C05455=1036.004,-58.740,418.899,168.441,38.908,157.287
C05456=1036.009,-58.491,418.887,168.443,38.908,157.287
C05457=1036.015,-58.241,418.875,168.446,38.907,157.287
C05458=1036.022,-57.992,418.863,168.448,38.907,157.287
C05459=1036.028,-57.742,418.850,168.451,38.906,157.287
C05460=1036.034,-57.492,418.839,168.453,38.906,157.287
C05461=1036.041,-57.242,418.827,168.456,38.906,157.287
C05462=1036.046,-56.993,418.815,168.458,38.905,157.287
C05463=1036.053,-56.743,418.803,168.461,38.905,157.287
C05464=1036.060,-56.494,418.791,168.464,38.904,157.287
C05465=1036.066,-56.248,418.779,168.466,38.904,157.287
C05466=1036.072,-56.003,418.767,168.469,38.904,157.287
C05467=1036.078,-55.758,418.755,168.470,38.903,157.287
C05468=1036.084,-55.512,418.743,168.473,38.903,157.287
C05469=1036.090,-55.268,418.731,168.475,38.902,157.286
C05470=1036.097,-55.022,418.720,168.478,38.902,157.287
C05471=1036.103,-54.777,418.707,168.480,38.902,157.287
C05472=1036.109,-54.531,418.696,168.483,38.901,157.286
C05473=1036.115,-54.282,418.684,168.485,38.901,157.287
C05474=1036.122,-54.032,418.672,168.488,38.901,157.287
C05475=1036.128,-53.782,418.659,168.490,38.900,157.286
C05476=1036.135,-53.533,418.647,168.493,38.900,157.287
C05477=1036.141,-53.283,418.635,168.495,38.899,157.286
C05478=1036.147,-53.033,418.623,168.498,38.899,157.286
C05479=1036.154,-52.784,418.611,168.500,38.899,157.287
C05480=1036.160,-52.534,418.599,168.503,38.898,157.286
C05481=1036.168,-52.244,418.584,168.506,38.898,157.286
C05482=1036.174,-51.954,418.570,168.509,38.897,157.286
C05483=1036.182,-51.664,418.556,168.512,38.897,157.286
C05484=1036.190,-51.373,418.541,168.515,38.896,157.286
C05485=1036.197,-51.124,418.529,168.517,38.896,157.286
C05486=1036.203,-50.874,418.517,168.520,38.895,157.286
C05487=1036.209,-50.624,418.505,168.522,38.895,157.286
C05488=1036.216,-50.375,418.493,168.525,38.894,157.286
C05489=1036.222,-50.125,418.480,168.527,38.894,157.286
C05490=1036.228,-49.876,418.467,168.530,38.894,157.287
C05491=1036.234,-49.626,418.454,168.532,38.894,157.287
C05492=1036.240,-49.377,418.443,168.535,38.894,157.287
C05493=1036.246,-49.127,418.430,168.537,38.893,157.287
C05494=1036.252,-48.878,418.417,168.539,38.893,157.287
C05495=1036.259,-48.628,418.405,168.542,38.893,157.287
C05496=1036.265,-48.378,418.393,168.544,38.893,157.287
C05497=1036.270,-48.129,418.380,168.547,38.892,157.287
C05498=1036.277,-47.880,418.367,168.549,38.892,157.287
C05499=1036.283,-47.630,418.355,168.552,38.892,157.287
C05500=1036.289,-47.380,418.342,168.554,38.892,157.287
C05501=1036.295,-47.131,418.329,168.557,38.891,157.287
C05502=1036.302,-46.881,418.317,168.559,38.891,157.287
C05503=1036.308,-46.631,418.304,168.562,38.891,157.287
C05504=1036.314,-46.382,418.291,168.564,38.891,157.287
C05505=1036.320,-46.132,418.279,168.566,38.891,157.287
C05506=1036.327,-45.882,418.267,168.569,38.890,157.287
C05507=1036.333,-45.633,418.253,168.571,38.890,157.287
C05508=1036.339,-45.383,418.241,168.574,38.889,157.287
C05509=1036.345,-45.134,418.229,168.576,38.889,157.287
C05510=1036.352,-44.884,418.215,168.579,38.889,157.287
C05511=1036.358,-44.634,418.203,168.581,38.889,157.287
C05512=1036.364,-44.385,418.189,168.584,38.889,157.287
C05513=1036.371,-44.135,418.177,168.586,38.889,157.287
C05514=1036.377,-43.885,418.165,168.588,38.889,157.287
C05515=1036.383,-43.636,418.152,168.591,38.888,157.287
C05516=1036.389,-43.386,418.139,168.593,38.888,157.287
C05517=1036.396,-43.137,418.126,168.596,38.887,157.287
C05518=1036.402,-42.887,418.114,168.598,38.887,157.287
C05519=1036.408,-42.638,418.101,168.601,38.887,157.287
C05520=1036.414,-42.388,418.088,168.603,38.887,157.287
C05521=1036.421,-42.139,418.075,168.606,38.887,157.287
C05522=1036.428,-41.888,418.062,168.608,38.887,157.287
C05523=1036.434,-41.639,418.049,168.610,38.887,157.287
C05524=1036.440,-41.389,418.037,168.613,38.886,157.287
C05525=1036.446,-41.140,418.023,168.615,38.886,157.287
C05526=1036.453,-40.890,418.011,168.618,38.885,157.287
C05527=1036.459,-40.641,417.998,168.620,38.885,157.287
C05528=1036.465,-40.391,417.986,168.623,38.885,157.287
C05529=1036.471,-40.141,417.972,168.625,38.885,157.287
C05530=1036.478,-39.892,417.960,168.627,38.885,157.287
C05531=1036.484,-39.642,417.947,168.630,38.885,157.288
C05532=1036.490,-39.393,417.934,168.632,38.885,157.288
C05533=1036.496,-39.143,417.921,168.635,38.884,157.287
C05534=1036.502,-38.893,417.908,168.637,38.884,157.288
C05535=1036.510,-38.644,417.895,168.640,38.883,157.288
C05536=1036.515,-38.394,417.881,168.642,38.883,157.288
C05537=1036.521,-38.144,417.869,168.644,38.883,157.288
C05538=1036.528,-37.895,417.856,168.647,38.883,157.288
C05539=1036.534,-37.646,417.842,168.649,38.883,157.288
C05540=1036.540,-37.396,417.830,168.651,38.883,157.288
C05541=1036.546,-37.146,417.816,168.654,38.883,157.288
C05542=1036.553,-36.897,417.803,168.656,38.883,157.288
C05543=1036.559,-36.647,417.790,168.659,38.883,157.288
C05544=1036.565,-36.398,417.777,168.662,38.883,157.288
C05545=1036.572,-36.117,417.762,168.665,38.883,157.288
C05546=1036.580,-35.835,417.747,168.667,38.882,157.288
C05547=1036.586,-35.554,417.733,168.670,38.882,157.288
C05548=1036.593,-35.273,417.718,168.673,38.882,157.288
C05549=1036.600,-35.024,417.704,168.675,38.882,157.288
C05550=1036.606,-34.774,417.692,168.677,38.882,157.288
C05551=1036.612,-34.524,417.678,168.680,38.882,157.288
C05552=1036.619,-34.275,417.665,168.682,38.882,157.288
C05553=1036.625,-34.026,417.652,168.684,38.881,157.288
C05554=1036.631,-33.776,417.639,168.687,38.881,157.288
C05555=1036.638,-33.526,417.625,168.689,38.881,157.288
C05556=1036.644,-33.277,417.612,168.692,38.881,157.289
C05557=1036.650,-33.027,417.599,168.694,38.881,157.289
C05558=1036.655,-32.778,417.585,168.696,38.881,157.289
C05559=1036.662,-32.528,417.571,168.699,38.880,157.289
C05560=1036.668,-32.278,417.559,168.701,38.880,157.289
C05561=1036.674,-32.029,417.546,168.703,38.880,157.289
C05562=1036.681,-31.780,417.532,168.706,38.880,157.289
C05563=1036.687,-31.530,417.519,168.708,38.880,157.289
C05564=1036.694,-31.280,417.505,168.710,38.880,157.289
C05565=1036.700,-31.031,417.492,168.713,38.880,157.289
C05566=1036.707,-30.781,417.479,168.715,38.880,157.289
C05567=1036.713,-30.532,417.465,168.717,38.880,157.289
C05568=1036.719,-30.283,417.452,168.720,38.880,157.289
C05569=1036.726,-30.032,417.439,168.722,38.880,157.289
C05570=1036.732,-29.783,417.426,168.725,38.880,157.289
C05571=1036.738,-29.533,417.413,168.727,38.879,157.289
C05572=1036.745,-29.283,417.399,168.729,38.879,157.289
C05573=1036.751,-29.034,417.386,168.732,38.879,157.289
C05574=1036.757,-28.785,417.372,168.734,38.879,157.289
C05575=1036.763,-28.535,417.358,168.736,38.879,157.289
C05576=1036.770,-28.285,417.345,168.739,38.879,157.289
C05577=1036.776,-28.036,417.332,168.741,38.879,157.289
C05578=1036.783,-27.786,417.318,168.743,38.878,157.289
C05579=1036.789,-27.537,417.305,168.746,38.878,157.289
C05580=1036.796,-27.287,417.291,168.748,38.878,157.290
C05581=1036.802,-27.038,417.278,168.750,38.878,157.290
C05582=1036.807,-26.788,417.264,168.753,38.878,157.290
C05583=1036.814,-26.538,417.250,168.755,38.878,157.290
C05584=1036.820,-26.289,417.237,168.757,38.878,157.290
C05585=1036.826,-26.039,417.223,168.761,38.878,157.290
C05586=1036.833,-25.789,417.209,168.763,38.878,157.290
C05587=1036.839,-25.541,417.196,168.765,38.878,157.290
C05588=1036.846,-25.291,417.182,168.767,38.878,157.290
C05589=1036.851,-25.041,417.168,168.770,38.878,157.290
C05590=1036.858,-24.792,417.155,168.772,38.878,157.290
C05591=1036.865,-24.542,417.141,168.774,38.878,157.290
C05592=1036.870,-24.292,417.127,168.777,38.878,157.290
C05593=1036.876,-24.043,417.114,168.779,38.878,157.290
C05594=1036.883,-23.793,417.099,168.781,38.878,157.290
C05595=1036.889,-23.544,417.086,168.783,38.878,157.290
C05596=1036.896,-23.294,417.072,168.786,38.878,157.290
C05597=1036.901,-23.045,417.058,168.788,38.878,157.290
C05598=1036.908,-22.795,417.045,168.790,38.878,157.291
C05599=1036.914,-22.546,417.031,168.793,38.878,157.291
C05600=1036.920,-22.296,417.017,168.795,38.878,157.291
C05601=1036.927,-22.046,417.003,168.797,38.878,157.291
C05602=1036.933,-21.797,416.990,168.799,38.878,157.291
C05603=1036.939,-21.548,416.975,168.802,38.877,157.291
C05604=1036.946,-21.298,416.962,168.804,38.878,157.291
C05605=1036.952,-21.048,416.948,168.806,38.878,157.291
C05606=1036.958,-20.799,416.934,168.809,38.878,157.291
C05607=1036.965,-20.549,416.920,168.811,38.878,157.291
C05608=1036.971,-20.300,416.907,168.813,38.877,157.291
C05609=1036.979,-20.018,416.890,168.817,38.878,157.291
C05610=1036.985,-19.736,416.875,168.819,38.878,157.291
C05611=1036.992,-19.454,416.859,168.822,38.878,157.291
C05612=1036.999,-19.172,416.843,168.824,38.877,157.291
C05613=1037.006,-18.923,416.829,168.827,38.877,157.291
C05614=1037.013,-18.673,416.816,168.829,38.878,157.292
C05615=1037.018,-18.424,416.802,168.831,38.878,157.292
C05616=1037.025,-18.174,416.787,168.833,38.878,157.292
C05617=1037.031,-17.925,416.774,168.836,38.877,157.292
C05618=1037.038,-17.675,416.760,168.838,38.877,157.292
C05619=1037.044,-17.426,416.746,168.840,38.877,157.292
C05620=1037.050,-17.176,416.732,168.843,38.878,157.292
C05621=1037.056,-16.927,416.718,168.845,38.877,157.292
C05622=1037.063,-16.677,416.704,168.847,38.877,157.292
C05623=1037.070,-16.427,416.690,168.849,38.877,157.292
C05624=1037.076,-16.178,416.676,168.852,38.877,157.292
C05625=1037.082,-15.928,416.662,168.854,38.878,157.292
C05626=1037.089,-15.680,416.648,168.856,38.877,157.292
C05627=1037.095,-15.430,416.634,168.858,38.877,157.292
C05628=1037.101,-15.180,416.620,168.861,38.877,157.292
C05629=1037.107,-14.930,416.605,168.863,38.878,157.292
C05630=1037.114,-14.681,416.592,168.865,38.877,157.293
C05631=1037.120,-14.431,416.577,168.867,38.877,157.293
C05632=1037.127,-14.182,416.563,168.870,38.878,157.293
C05633=1037.133,-13.933,416.549,168.873,38.878,157.293
C05634=1037.139,-13.683,416.534,168.875,38.878,157.293
C05635=1037.145,-13.434,416.521,168.877,38.878,157.293
C05636=1037.152,-13.184,416.506,168.879,38.878,157.293
C05637=1037.157,-12.934,416.492,168.882,38.878,157.293
C05638=1037.164,-12.685,416.477,168.884,38.878,157.293
C05639=1037.170,-12.435,416.463,168.886,38.878,157.293
C05640=1037.176,-12.186,416.449,168.888,38.878,157.293
C05641=1037.183,-11.936,416.434,168.890,38.879,157.293
C05642=1037.189,-11.687,416.420,168.893,38.878,157.293
C05643=1037.196,-11.438,416.406,168.895,38.878,157.293
C05644=1037.202,-11.188,416.391,168.897,38.878,157.293
C05645=1037.208,-10.938,416.377,168.899,38.879,157.294
C05646=1037.215,-10.689,416.363,168.901,38.879,157.294
C05647=1037.221,-10.439,416.349,168.904,38.878,157.294
C05648=1037.227,-10.190,416.334,168.906,38.879,157.294
C05649=1037.234,-9.940,416.320,168.908,38.879,157.294
C05650=1037.239,-9.691,416.306,168.910,38.879,157.294
C05651=1037.246,-9.441,416.291,168.913,38.879,157.294
C05652=1037.253,-9.192,416.277,168.916,38.879,157.294
C05653=1037.258,-8.943,416.262,168.918,38.879,157.294
C05654=1037.264,-8.693,416.248,168.920,38.879,157.294
C05655=1037.272,-8.443,416.233,168.922,38.879,157.294
C05656=1037.277,-8.194,416.219,168.924,38.879,157.294
C05657=1037.283,-7.944,416.205,168.927,38.880,157.295
C05658=1037.291,-7.695,416.190,168.929,38.880,157.295
C05659=1037.297,-7.445,416.175,168.931,38.879,157.295
C05660=1037.303,-7.196,416.161,168.933,38.880,157.295
C05661=1037.310,-6.946,416.147,168.935,38.880,157.295
C05662=1037.316,-6.696,416.132,168.938,38.880,157.295
C05663=1037.322,-6.447,416.118,168.940,38.880,157.295
C05664=1037.328,-6.198,416.103,168.942,38.880,157.295
C05665=1037.335,-5.948,416.089,168.944,38.880,157.295
C05666=1037.341,-5.698,416.074,168.946,38.880,157.295
C05667=1037.347,-5.449,416.059,168.949,38.880,157.295
C05668=1037.354,-5.200,416.045,168.951,38.880,157.295
C05669=1037.361,-4.950,416.030,168.953,38.880,157.295
C05670=1037.367,-4.701,416.015,168.956,38.881,157.295
C05671=1037.373,-4.451,416.002,168.958,38.880,157.296
C05672=1037.380,-4.202,415.987,168.960,38.880,157.296
C05673=1037.387,-3.918,415.971,168.963,38.881,157.296
C05674=1037.394,-3.635,415.954,168.965,38.881,157.296
C05675=1037.402,-3.351,415.937,168.968,38.881,157.296
C05676=1037.408,-3.067,415.920,168.970,38.881,157.296
C05677=1037.414,-2.818,415.905,168.972,38.881,157.296
C05678=1037.420,-2.569,415.890,168.975,38.881,157.296
C05679=1037.427,-2.319,415.875,168.977,38.882,157.296
C05680=1037.433,-2.069,415.861,168.979,38.882,157.296
C05681=1037.439,-1.820,415.846,168.981,38.882,157.296
C05682=1037.445,-1.571,415.831,168.983,38.882,157.297
C05683=1037.452,-1.321,415.816,168.985,38.883,157.297
C05684=1037.458,-1.071,415.801,168.987,38.882,157.297
C05685=1037.464,-0.823,415.787,168.990,38.883,157.297
C05686=1037.470,-0.573,415.772,168.993,38.883,157.297
C05687=1037.476,-0.323,415.757,168.995,38.883,157.297
C05688=1037.483,-0.074,415.742,168.997,38.883,157.297
C05689=1037.489,0.175,415.727,168.999,38.884,157.297
C05690=1037.495,0.425,415.712,169.001,38.884,157.297
C05691=1037.501,0.675,415.697,169.003,38.884,157.297
C05692=1037.508,0.924,415.682,169.005,38.884,157.297
C05693=1037.514,1.173,415.667,169.007,38.885,157.298
C05694=1037.520,1.422,415.652,169.009,38.884,157.298
C05695=1037.527,1.672,415.637,169.012,38.884,157.298
C05696=1037.533,1.922,415.622,169.014,38.885,157.298
C05697=1037.539,2.171,415.607,169.016,38.885,157.298
C05698=1037.546,2.421,415.592,169.019,38.885,157.298
C05699=1037.552,2.671,415.577,169.021,38.885,157.298
C05700=1037.558,2.920,415.563,169.023,38.886,157.298
C05701=1037.565,3.169,415.547,169.025,38.885,157.298
C05702=1037.571,3.418,415.532,169.027,38.886,157.298
C05703=1037.577,3.668,415.517,169.029,38.886,157.298
C05704=1037.584,3.918,415.502,169.032,38.886,157.299
C05705=1037.590,4.167,415.487,169.034,38.886,157.299
C05706=1037.595,4.417,415.472,169.036,38.887,157.299
C05707=1037.602,4.666,415.456,169.038,38.887,157.299
C05708=1037.608,4.915,415.441,169.040,38.887,157.299
C05709=1037.615,5.165,415.427,169.042,38.887,157.299
C05710=1037.621,5.415,415.412,169.044,38.888,157.299
C05711=1037.627,5.664,415.397,169.046,38.887,157.299
C05712=1037.634,5.913,415.381,169.049,38.888,157.299
C05713=1037.641,6.163,415.366,169.052,38.888,157.299
C05714=1037.647,6.413,415.351,169.054,38.888,157.299
C05715=1037.653,6.662,415.337,169.056,38.888,157.300
C05716=1037.659,6.911,415.321,169.058,38.888,157.300
C05717=1037.666,7.160,415.306,169.060,38.889,157.300
C05718=1037.672,7.410,415.291,169.062,38.888,157.300
C05719=1037.679,7.660,415.276,169.064,38.889,157.300
C05720=1037.685,7.909,415.260,169.066,38.889,157.300
C05721=1037.691,8.159,415.245,169.068,38.889,157.300
C05722=1037.697,8.408,415.230,169.070,38.889,157.300
C05723=1037.704,8.657,415.214,169.073,38.890,157.300
C05724=1037.710,8.907,415.199,169.075,38.890,157.300
C05725=1037.717,9.157,415.184,169.077,38.889,157.300
C05726=1037.723,9.406,415.169,169.080,38.890,157.301
C05727=1037.730,9.655,415.154,169.082,38.890,157.301
C05728=1037.736,9.905,415.139,169.084,38.890,157.301
C05729=1037.743,10.154,415.123,169.086,38.890,157.301
C05730=1037.749,10.404,415.108,169.088,38.891,157.301
C05731=1037.756,10.653,415.093,169.090,38.891,157.301
C05732=1037.762,10.902,415.078,169.092,38.891,157.301
C05733=1037.768,11.152,415.062,169.095,38.891,157.301
C05734=1037.774,11.402,415.047,169.097,38.891,157.301
C05735=1037.781,11.651,415.031,169.099,38.891,157.301
C05736=1037.787,11.901,415.016,169.101,38.891,157.301
C05737=1037.795,12.186,414.999,169.103,38.892,157.301
C05738=1037.802,12.471,414.981,169.106,38.892,157.302
C05739=1037.810,12.757,414.964,169.108,38.892,157.302
C05740=1037.817,13.042,414.946,169.110,38.892,157.302
C05741=1037.824,13.291,414.931,169.114,38.892,157.302
C05742=1037.830,13.541,414.916,169.116,38.892,157.302
C05743=1037.836,13.790,414.900,169.118,38.893,157.302
C05744=1037.843,14.040,414.885,169.120,38.893,157.302
C05745=1037.849,14.289,414.869,169.122,38.893,157.302
C05746=1037.856,14.538,414.854,169.124,38.893,157.302
C05747=1037.862,14.788,414.838,169.126,38.894,157.302
C05748=1037.868,15.037,414.823,169.128,38.893,157.302
C05749=1037.875,15.287,414.807,169.130,38.894,157.303
C05750=1037.880,15.536,414.792,169.132,38.895,157.303
C05751=1037.887,15.786,414.776,169.134,38.894,157.303
C05752=1037.893,16.035,414.760,169.136,38.895,157.303
C05753=1037.899,16.285,414.745,169.138,38.895,157.303
C05754=1037.906,16.534,414.729,169.141,38.895,157.303
C05755=1037.912,16.784,414.714,169.143,38.895,157.303
C05756=1037.918,17.033,414.698,169.145,38.896,157.303
C05757=1037.925,17.282,414.682,169.147,38.896,157.303
C05758=1037.931,17.532,414.667,169.149,38.896,157.304
C05759=1037.937,17.781,414.651,169.151,38.897,157.304
C05760=1037.943,18.030,414.635,169.153,38.896,157.304
C05761=1037.950,18.280,414.619,169.156,38.897,157.304
C05762=1037.957,18.529,414.604,169.158,38.897,157.304
C05763=1037.963,18.779,414.588,169.160,38.897,157.304
C05764=1037.969,19.028,414.573,169.162,38.897,157.304
C05765=1037.976,19.277,414.557,169.164,38.898,157.304
C05766=1037.982,19.527,414.541,169.167,38.898,157.304
C05767=1037.988,19.776,414.526,169.169,38.898,157.304
C05768=1037.994,20.026,414.509,169.171,38.899,157.305
C05769=1038.001,20.275,414.494,169.173,38.899,157.305
C05770=1038.007,20.525,414.478,169.175,38.899,157.305
C05771=1038.014,20.775,414.462,169.177,38.900,157.305
C05772=1038.020,21.024,414.446,169.179,38.899,157.305
C05773=1038.027,21.273,414.430,169.181,38.900,157.305
C05774=1038.033,21.522,414.414,169.183,38.900,157.305
C05775=1038.039,21.772,414.399,169.185,38.900,157.305
C05776=1038.045,22.021,414.383,169.187,38.901,157.305
C05777=1038.052,22.270,414.367,169.189,38.901,157.305
C05778=1038.058,22.520,414.351,169.192,38.901,157.306
C05779=1038.065,22.769,414.335,169.194,38.902,157.306
C05780=1038.071,23.019,414.319,169.196,38.902,157.306
C05781=1038.077,23.268,414.304,169.198,38.902,157.306
C05782=1038.083,23.518,414.287,169.200,38.902,157.306
C05783=1038.090,23.767,414.272,169.202,38.903,157.306
C05784=1038.096,24.016,414.256,169.204,38.903,157.306
C05785=1038.102,24.265,414.239,169.206,38.903,157.306
C05786=1038.109,24.516,414.224,169.208,38.904,157.306
C05787=1038.115,24.765,414.208,169.210,38.903,157.307
C05788=1038.121,25.014,414.192,169.212,38.904,157.307
C05789=1038.127,25.264,414.176,169.215,38.904,157.307
C05790=1038.134,25.513,414.160,169.217,38.904,157.307
C05791=1038.141,25.763,414.144,169.219,38.905,157.307
C05792=1038.147,26.012,414.128,169.221,38.905,157.307
C05793=1038.153,26.261,414.112,169.223,38.905,157.307
C05794=1038.159,26.510,414.095,169.225,38.906,157.307
C05795=1038.166,26.759,414.080,169.227,38.906,157.307
C05796=1038.172,27.009,414.063,169.229,38.906,157.308
C05797=1038.179,27.258,414.047,169.231,38.906,157.308
C05798=1038.185,27.508,414.031,169.233,38.907,157.308
C05799=1038.191,27.758,414.016,169.235,38.907,157.308
C05800=1038.198,28.008,414.000,169.237,38.907,157.308
C05801=1038.205,28.294,413.981,169.240,38.907,157.308
C05802=1038.212,28.580,413.962,169.243,38.908,157.308
C05803=1038.219,28.867,413.944,169.245,38.908,157.308
C05804=1038.226,29.153,413.925,169.247,38.908,157.308
C05805=1038.233,29.404,413.908,169.249,38.909,157.309
C05806=1038.239,29.653,413.892,169.251,38.909,157.309
C05807=1038.246,29.902,413.877,169.253,38.910,157.309
C05808=1038.252,30.151,413.860,169.255,38.910,157.309
C05809=1038.258,30.401,413.844,169.257,38.910,157.309
C05810=1038.264,30.650,413.827,169.260,38.911,157.309
C05811=1038.271,30.899,413.811,169.262,38.911,157.309
C05812=1038.277,31.148,413.795,169.264,38.911,157.309
C05813=1038.284,31.398,413.778,169.266,38.912,157.310
C05814=1038.290,31.648,413.762,169.268,38.912,157.310
C05815=1038.296,31.897,413.746,169.270,38.912,157.310
C05816=1038.302,32.146,413.730,169.272,38.913,157.310
C05817=1038.309,32.396,413.713,169.274,38.912,157.310
C05818=1038.315,32.645,413.696,169.276,38.913,157.310
C05819=1038.321,32.894,413.680,169.278,38.913,157.310
C05820=1038.327,33.144,413.664,169.280,38.913,157.310
C05821=1038.334,33.393,413.648,169.283,38.914,157.310
C05822=1038.340,33.643,413.632,169.285,38.914,157.311
C05823=1038.346,33.891,413.615,169.287,38.915,157.311
C05824=1038.353,34.142,413.598,169.289,38.915,157.311
C05825=1038.360,34.391,413.582,169.291,38.915,157.311
C05826=1038.366,34.640,413.566,169.293,38.916,157.311
C05827=1038.372,34.890,413.549,169.295,38.916,157.311
C05828=1038.378,35.139,413.533,169.297,38.916,157.311
C05829=1038.384,35.388,413.516,169.299,38.917,157.311
C05830=1038.392,35.638,413.500,169.301,38.917,157.311
C05831=1038.398,35.887,413.484,169.303,38.917,157.312
C05832=1038.404,36.136,413.467,169.305,38.917,157.312
C05833=1038.410,36.386,413.450,169.307,38.918,157.312
C05834=1038.416,36.635,413.434,169.309,38.918,157.312
C05835=1038.422,36.885,413.418,169.311,38.918,157.312
C05836=1038.430,37.134,413.401,169.313,38.918,157.312
C05837=1038.436,37.383,413.385,169.315,38.919,157.312
C05838=1038.442,37.633,413.368,169.317,38.920,157.312
C05839=1038.449,37.882,413.351,169.319,38.919,157.312
C05840=1038.455,38.131,413.335,169.321,38.920,157.313
C05841=1038.461,38.381,413.318,169.323,38.920,157.313
C05842=1038.467,38.630,413.301,169.326,38.921,157.313
C05843=1038.473,38.879,413.285,169.328,38.921,157.313
C05844=1038.480,39.129,413.268,169.330,38.921,157.313
C05845=1038.486,39.378,413.252,169.332,38.922,157.313
C05846=1038.492,39.627,413.235,169.334,38.922,157.313
C05847=1038.499,39.877,413.218,169.336,38.922,157.313
C05848=1038.505,40.126,413.202,169.338,38.923,157.314
C05849=1038.512,40.376,413.184,169.340,38.923,157.314
C05850=1038.517,40.625,413.168,169.342,38.924,157.314
C05851=1038.523,40.874,413.151,169.344,38.924,157.314
C05852=1038.530,41.124,413.134,169.346,38.924,157.314
C05853=1038.536,41.373,413.118,169.348,38.925,157.314
C05854=1038.543,41.623,413.100,169.350,38.925,157.314
C05855=1038.549,41.872,413.084,169.352,38.926,157.315
C05856=1038.555,42.121,413.067,169.354,38.926,157.315
C05857=1038.561,42.371,413.050,169.356,38.926,157.315
C05858=1038.568,42.620,413.034,169.358,38.927,157.315
C05859=1038.574,42.870,413.017,169.360,38.927,157.315
C05860=1038.581,43.119,413.000,169.362,38.927,157.315
C05861=1038.586,43.368,412.984,169.365,38.928,157.315
C05862=1038.593,43.617,412.966,169.367,38.928,157.315
C05863=1038.599,43.866,412.949,169.369,38.929,157.315
C05864=1038.605,44.116,412.932,169.370,38.929,157.316
C05865=1038.612,44.403,412.913,169.373,38.930,157.316
C05866=1038.619,44.689,412.893,169.375,38.930,157.316
C05867=1038.626,44.976,412.873,169.377,38.931,157.316
C05868=1038.634,45.262,412.854,169.379,38.931,157.316
C05869=1038.640,45.512,412.837,169.382,38.932,157.316
C05870=1038.646,45.761,412.820,169.384,38.932,157.317
C05871=1038.653,46.010,412.802,169.386,38.932,157.317
C05872=1038.658,46.260,412.786,169.388,38.933,157.317
C05873=1038.664,46.509,412.769,169.390,38.933,157.317
C05874=1038.671,46.758,412.751,169.392,38.934,157.317
C05875=1038.676,47.008,412.734,169.394,38.934,157.317
C05876=1038.683,47.257,412.717,169.395,38.935,157.317
C05877=1038.690,47.506,412.700,169.398,38.935,157.318
C05878=1038.695,47.756,412.683,169.400,38.935,157.318
C05879=1038.702,48.005,412.666,169.402,38.936,157.318
C05880=1038.708,48.254,412.649,169.404,38.936,157.318
C05881=1038.715,48.503,412.632,169.406,38.937,157.318
C05882=1038.721,48.754,412.614,169.408,38.937,157.318
C05883=1038.727,49.002,412.597,169.410,38.938,157.318
C05884=1038.734,49.252,412.580,169.412,38.938,157.318
C05885=1038.739,49.501,412.563,169.414,38.938,157.319
C05886=1038.746,49.751,412.546,169.416,38.939,157.319
C05887=1038.752,50.000,412.529,169.418,38.939,157.319
C05888=1038.758,50.249,412.511,169.420,38.940,157.319
C05889=1038.764,50.498,412.494,169.422,38.940,157.319
C05890=1038.771,50.748,412.477,169.424,38.941,157.319
C05891=1038.776,50.997,412.460,169.426,38.941,157.319
C05892=1038.783,51.247,412.443,169.428,38.941,157.319
C05893=1038.790,51.495,412.426,169.430,38.942,157.320
C05894=1038.796,51.745,412.408,169.432,38.942,157.320
C05895=1038.802,51.994,412.391,169.435,38.943,157.320
C05896=1038.808,52.244,412.374,169.436,38.943,157.320
C05897=1038.814,52.493,412.356,169.438,38.943,157.320
C05898=1038.821,52.742,412.339,169.440,38.944,157.320
C05899=1038.828,52.992,412.322,169.442,38.944,157.320
C05900=1038.833,53.241,412.304,169.444,38.945,157.321
C05901=1038.840,53.490,412.287,169.446,38.945,157.321
C05902=1038.845,53.740,412.270,169.448,38.945,157.321
C05903=1038.852,53.989,412.253,169.450,38.946,157.321
C05904=1038.858,54.238,412.236,169.453,38.946,157.321
C05905=1038.865,54.488,412.218,169.455,38.947,157.321
C05906=1038.871,54.737,412.200,169.457,38.947,157.321
C05907=1038.878,54.986,412.183,169.458,38.947,157.321
C05908=1038.884,55.236,412.166,169.460,38.948,157.322
C05909=1038.890,55.484,412.149,169.462,38.948,157.322
C05910=1038.897,55.734,412.131,169.464,38.949,157.322
C05911=1038.903,55.984,412.113,169.466,38.949,157.322
C05912=1038.909,56.232,412.096,169.468,38.949,157.322
C05913=1038.916,56.482,412.079,169.471,38.949,157.322
C05914=1038.922,56.731,412.061,169.473,38.950,157.322
C05915=1038.929,56.980,412.044,169.475,38.950,157.322
C05916=1038.934,57.231,412.027,169.477,38.951,157.323
C05917=1038.941,57.479,412.010,169.479,38.951,157.323
C05918=1038.947,57.729,411.993,169.480,38.951,157.323
C05919=1038.954,57.978,411.975,169.482,38.952,157.323
C05920=1038.960,58.227,411.958,169.484,38.952,157.323
C05921=1038.967,58.477,411.940,169.486,38.952,157.323
C05922=1038.973,58.726,411.922,169.488,38.953,157.323
C05923=1038.979,58.974,411.905,169.491,38.953,157.323
C05924=1038.985,59.224,411.887,169.493,38.954,157.324
C05925=1038.992,59.474,411.869,169.495,38.954,157.324
C05926=1038.999,59.723,411.852,169.497,38.954,157.324
C05927=1039.005,59.972,411.834,169.499,38.955,157.324
C05928=1039.012,60.221,411.817,169.501,38.955,157.324
C05929=1039.019,60.507,411.797,169.503,38.956,157.324
C05930=1039.026,60.794,411.777,169.505,38.956,157.324
C05931=1039.034,61.081,411.757,169.507,38.956,157.324
C05932=1039.041,61.367,411.737,169.510,38.957,157.325
C05933=1039.047,61.616,411.719,169.512,38.957,157.325
C05934=1039.054,61.866,411.701,169.514,38.958,157.325
C05935=1039.060,62.115,411.684,169.516,38.958,157.325
C05936=1039.067,62.364,411.667,169.518,38.958,157.325
C05937=1039.073,62.613,411.648,169.520,38.959,157.325
C05938=1039.080,62.863,411.631,169.522,38.959,157.325
C05939=1039.086,63.112,411.613,169.524,38.959,157.325
C05940=1039.092,63.361,411.596,169.526,38.959,157.326
C05941=1039.099,63.610,411.579,169.529,38.960,157.326
C05942=1039.105,63.860,411.561,169.531,38.961,157.326
C05943=1039.111,64.109,411.543,169.533,38.961,157.326
C05944=1039.118,64.358,411.525,169.534,38.961,157.326
C05945=1039.124,64.608,411.507,169.536,38.961,157.326
C05946=1039.130,64.857,411.489,169.538,38.962,157.326
C05947=1039.137,65.106,411.472,169.540,38.963,157.327
C05948=1039.143,65.355,411.454,169.542,38.963,157.327
C05949=1039.149,65.605,411.436,169.544,38.964,157.327
C05950=1039.155,65.854,411.419,169.547,38.964,157.327
C05951=1039.162,66.103,411.400,169.549,38.965,157.327
C05952=1039.168,66.353,411.382,169.551,38.965,157.327
C05953=1039.175,66.602,411.365,169.552,38.965,157.327
C05954=1039.181,66.851,411.346,169.554,38.965,157.328
C05955=1039.187,67.100,411.329,169.556,38.966,157.328
C05956=1039.194,67.350,411.311,169.558,38.967,157.328
C05957=1039.200,67.599,411.293,169.560,38.967,157.328
C05958=1039.206,67.849,411.275,169.563,38.968,157.328
C05959=1039.212,68.098,411.257,169.565,38.968,157.328
C05960=1039.219,68.346,411.239,169.567,38.969,157.328
C05961=1039.225,68.596,411.221,169.568,38.968,157.328
C05962=1039.231,68.845,411.203,169.570,38.969,157.329
C05963=1039.237,69.095,411.185,169.572,38.970,157.329
C05964=1039.244,69.344,411.168,169.574,38.970,157.329
C05965=1039.250,69.593,411.149,169.576,38.971,157.329
C05966=1039.256,69.843,411.131,169.579,38.971,157.329
C05967=1039.263,70.092,411.112,169.581,38.972,157.329
C05968=1039.268,70.341,411.095,169.583,38.972,157.330
C05969=1039.275,70.590,411.076,169.584,38.973,157.330
C05970=1039.281,70.839,411.059,169.586,38.973,157.330
C05971=1039.288,71.088,411.040,169.588,38.974,157.330
C05972=1039.294,71.338,411.022,169.590,38.974,157.330
C05973=1039.300,71.587,411.005,169.592,38.975,157.330
C05974=1039.306,71.836,410.986,169.595,38.975,157.330
C05975=1039.312,72.085,410.967,169.597,38.975,157.330
C05976=1039.319,72.335,410.950,169.599,38.976,157.331
C05977=1039.325,72.584,410.931,169.600,38.976,157.331
C05978=1039.332,72.834,410.914,169.602,38.977,157.331
C05979=1039.338,73.082,410.895,169.604,38.977,157.331
C05980=1039.344,73.332,410.877,169.606,38.978,157.331
C05981=1039.350,73.581,410.859,169.608,38.978,157.331
C05982=1039.356,73.831,410.841,169.611,38.979,157.332
C05983=1039.363,74.080,410.822,169.613,38.979,157.332
C05984=1039.369,74.330,410.804,169.615,38.980,157.332
C05985=1039.375,74.578,410.786,169.616,38.980,157.332
C05986=1039.381,74.827,410.767,169.618,38.981,157.332
C05987=1039.387,75.077,410.749,169.620,38.981,157.332
C05988=1039.394,75.326,410.731,169.622,38.982,157.332
C05989=1039.400,75.576,410.713,169.624,38.982,157.333
C05990=1039.407,75.825,410.695,169.626,38.982,157.333
C05991=1039.413,76.074,410.676,169.629,38.983,157.333
C05992=1039.419,76.323,410.658,169.631,38.983,157.333
C05993=1039.426,76.609,410.637,169.633,38.984,157.333
C05994=1039.434,76.895,410.616,169.635,38.984,157.333
C05995=1039.441,77.181,410.594,169.637,38.985,157.333
C05996=1039.448,77.467,410.573,169.639,38.985,157.334
C05997=1039.454,77.716,410.556,169.641,38.986,157.334
C05998=1039.461,77.966,410.537,169.644,38.986,157.334
C05999=1039.467,78.215,410.518,169.646,38.987,157.334
C06000=1039.473,78.465,410.500,169.648,38.987,157.334
C06001=1039.479,78.714,410.481,169.650,38.988,157.334
C06002=1039.485,78.963,410.462,169.651,38.988,157.335
C06003=1039.492,79.212,410.444,169.653,38.989,157.335
C06004=1039.498,79.461,410.426,169.655,38.990,157.335
C06005=1039.504,79.710,410.408,169.658,38.990,157.335
C06006=1039.510,79.960,410.388,169.660,38.991,157.335
C06007=1039.516,80.209,410.370,169.662,38.992,157.335
C06008=1039.522,80.458,410.351,169.664,38.992,157.336
C06009=1039.529,80.707,410.332,169.665,38.993,157.336
C06010=1039.535,80.957,410.314,169.667,38.993,157.336
C06011=1039.541,81.206,410.296,169.669,38.994,157.336
C06012=1039.547,81.455,410.277,169.672,38.994,157.336
C06013=1039.553,81.705,410.258,169.674,38.995,157.336
C06014=1039.560,81.954,410.239,169.676,38.995,157.337
C06015=1039.566,82.203,410.221,169.678,38.996,157.337
C06016=1039.573,82.452,410.202,169.679,38.996,157.337
C06017=1039.578,82.701,410.184,169.681,38.997,157.337
C06018=1039.584,82.950,410.165,169.683,38.997,157.337
C06019=1039.590,83.199,410.146,169.686,38.998,157.337
C06020=1039.597,83.449,410.128,169.688,38.998,157.337
C06021=1039.603,83.698,410.109,169.690,38.999,157.338
C06022=1039.609,83.947,410.090,169.692,38.999,157.338
C06023=1039.615,84.196,410.071,169.694,39.000,157.338
C06024=1039.622,84.445,410.053,169.695,39.000,157.338
C06025=1039.628,84.695,410.034,169.697,39.001,157.338
C06026=1039.635,84.944,410.015,169.699,39.001,157.338
C06027=1039.640,85.193,409.996,169.702,39.002,157.339
C06028=1039.647,85.442,409.977,169.704,39.002,157.339
C06029=1039.653,85.691,409.959,169.706,39.003,157.339
C06030=1039.660,85.940,409.940,169.708,39.003,157.339
C06031=1039.666,86.190,409.922,169.710,39.004,157.339
C06032=1039.671,86.440,409.903,169.711,39.004,157.339
C06033=1039.678,86.689,409.884,169.713,39.005,157.339
C06034=1039.685,86.937,409.865,169.716,39.005,157.340
C06035=1039.692,87.187,409.846,169.718,39.005,157.340
C06036=1039.697,87.436,409.827,169.720,39.006,157.340
C06037=1039.704,87.686,409.808,169.722,39.006,157.340
C06038=1039.710,87.935,409.789,169.724,39.007,157.340
C06039=1039.717,88.184,409.771,169.726,39.007,157.340
C06040=1039.723,88.433,409.752,169.728,39.008,157.340
C06041=1039.729,88.682,409.733,169.729,39.008,157.341
C06042=1039.735,88.932,409.714,169.731,39.009,157.341
C06043=1039.742,89.181,409.696,169.734,39.009,157.341
C06044=1039.748,89.430,409.677,169.736,39.010,157.341
C06045=1039.754,89.679,409.658,169.738,39.010,157.341
C06046=1039.760,89.928,409.639,169.740,39.011,157.341
C06047=1039.766,90.177,409.620,169.742,39.011,157.341
C06048=1039.772,90.427,409.601,169.744,39.012,157.342
C06049=1039.779,90.675,409.582,169.746,39.012,157.342
C06050=1039.785,90.926,409.562,169.748,39.013,157.342
C06051=1039.792,91.175,409.544,169.750,39.014,157.342
C06052=1039.797,91.424,409.524,169.752,39.015,157.342
C06053=1039.804,91.673,409.506,169.754,39.015,157.343
C06054=1039.810,91.922,409.486,169.756,39.016,157.343
C06055=1039.816,92.171,409.467,169.758,39.016,157.343
C06056=1039.822,92.421,409.448,169.760,39.017,157.343
C06057=1039.829,92.707,409.426,169.763,39.017,157.343
C06058=1039.836,92.993,409.404,169.765,39.018,157.343
C06059=1039.844,93.279,409.382,169.767,39.019,157.344
C06060=1039.850,93.564,409.360,169.769,39.019,157.344
C06061=1039.857,93.814,409.341,169.771,39.020,157.344
C06062=1039.863,94.063,409.322,169.773,39.020,157.344
C06063=1039.869,94.312,409.302,169.776,39.021,157.344
C06064=1039.876,94.561,409.283,169.778,39.021,157.344
C06065=1039.881,94.811,409.264,169.780,39.022,157.345
C06066=1039.888,95.059,409.245,169.781,39.022,157.345
C06067=1039.894,95.308,409.225,169.783,39.023,157.345
C06068=1039.900,95.558,409.207,169.785,39.023,157.345
C06069=1039.907,95.807,409.187,169.787,39.024,157.345
C06070=1039.913,96.056,409.168,169.790,39.025,157.345
C06071=1039.919,96.306,409.149,169.792,39.026,157.346
C06072=1039.925,96.554,409.129,169.794,39.026,157.346
C06073=1039.931,96.804,409.110,169.796,39.027,157.346
C06074=1039.937,97.053,409.091,169.797,39.027,157.346
C06075=1039.944,97.302,409.071,169.799,39.028,157.346
C06076=1039.950,97.552,409.052,169.801,39.028,157.346
C06077=1039.956,97.801,409.033,169.804,39.029,157.347
C06078=1039.962,98.050,409.013,169.806,39.029,157.347
C06079=1039.969,98.299,408.995,169.808,39.030,157.347
C06080=1039.975,98.548,408.975,169.810,39.030,157.347
C06081=1039.982,98.797,408.956,169.812,39.031,157.347
C06082=1039.987,99.047,408.936,169.814,39.031,157.347
C06083=1039.994,99.295,408.917,169.816,39.032,157.347
C06084=1040.000,99.545,408.898,169.818,39.032,157.348
C06085=1040.007,99.793,408.878,169.820,39.033,157.348
C06086=1040.013,100.043,408.859,169.822,39.033,157.348
C06087=1040.019,100.292,408.839,169.824,39.034,157.348
C06088=1040.025,100.541,408.820,169.826,39.034,157.348
C06089=1040.031,100.790,408.800,169.828,39.035,157.349
C06090=1040.037,101.040,408.781,169.830,39.036,157.349
C06091=1040.044,101.289,408.761,169.833,39.036,157.349
C06092=1040.050,101.538,408.742,169.834,39.037,157.349
C06093=1040.056,101.787,408.722,169.836,39.037,157.349
C06094=1040.062,102.036,408.702,169.838,39.038,157.349
C06095=1040.068,102.285,408.683,169.840,39.039,157.350
C06096=1040.074,102.535,408.662,169.842,39.040,157.350
C06097=1040.081,102.784,408.644,169.845,39.040,157.350
C06098=1040.087,103.033,408.624,169.847,39.041,157.350
C06099=1040.092,103.282,408.605,169.849,39.041,157.350
C06100=1040.099,103.532,408.584,169.851,39.042,157.350
C06101=1040.105,103.780,408.564,169.852,39.043,157.351
C06102=1040.111,104.030,408.545,169.854,39.043,157.351
C06103=1040.117,104.278,408.526,169.856,39.044,157.351
C06104=1040.123,104.527,408.506,169.859,39.044,157.351
C06105=1040.130,104.777,408.486,169.861,39.045,157.351
C06106=1040.136,105.026,408.466,169.863,39.045,157.351
C06107=1040.142,105.275,408.446,169.865,39.046,157.352
C06108=1040.149,105.525,408.427,169.867,39.047,157.352
C06109=1040.155,105.774,408.407,169.869,39.047,157.352
C06110=1040.161,106.022,408.387,169.871,39.048,157.352
C06111=1040.166,106.272,408.368,169.873,39.048,157.352
C06112=1040.173,106.521,408.348,169.875,39.049,157.352
C06113=1040.179,106.770,408.328,169.877,39.049,157.353
C06114=1040.186,107.019,408.308,169.879,39.050,157.353
C06115=1040.192,107.269,408.289,169.881,39.050,157.353
C06116=1040.198,107.518,408.269,169.883,39.052,157.353
C06117=1040.204,107.766,408.249,169.886,39.052,157.353
C06118=1040.210,108.015,408.229,169.888,39.053,157.354
C06119=1040.216,108.265,408.209,169.890,39.053,157.354
C06120=1040.223,108.514,408.190,169.892,39.054,157.354
C06121=1040.230,108.800,408.167,169.894,39.054,157.354
C06122=1040.237,109.086,408.145,169.896,39.055,157.354
C06123=1040.244,109.372,408.121,169.899,39.056,157.354
C06124=1040.251,109.658,408.098,169.901,39.056,157.355
C06125=1040.258,109.907,408.079,169.903,39.057,157.355
C06126=1040.264,110.156,408.059,169.905,39.057,157.355
C06127=1040.270,110.405,408.039,169.907,39.058,157.355
C06128=1040.276,110.654,408.019,169.909,39.059,157.355
C06129=1040.283,110.904,407.999,169.912,39.059,157.356
C06130=1040.289,111.153,407.979,169.914,39.060,157.356
C06131=1040.295,111.402,407.959,169.916,39.060,157.356
C06132=1040.301,111.651,407.939,169.918,39.061,157.356
C06133=1040.307,111.900,407.919,169.920,39.062,157.356
C06134=1040.313,112.149,407.899,169.921,39.063,157.356
C06135=1040.320,112.398,407.879,169.923,39.063,157.357
C06136=1040.326,112.647,407.859,169.926,39.064,157.357
C06137=1040.332,112.896,407.839,169.928,39.064,157.357
C06138=1040.338,113.146,407.818,169.930,39.065,157.357
C06139=1040.344,113.394,407.799,169.932,39.066,157.357
C06140=1040.351,113.644,407.778,169.934,39.066,157.357
C06141=1040.357,113.893,407.758,169.936,39.067,157.358
C06142=1040.362,114.142,407.738,169.939,39.068,157.358
C06143=1040.369,114.391,407.717,169.941,39.068,157.358
C06144=1040.375,114.640,407.697,169.943,39.069,157.358
C06145=1040.381,114.889,407.677,169.944,39.070,157.359
C06146=1040.387,115.139,407.657,169.946,39.071,157.359
C06147=1040.393,115.388,407.637,169.948,39.071,157.359
C06148=1040.399,115.636,407.617,169.951,39.071,157.359
C06149=1040.405,115.886,407.596,169.953,39.073,157.359
C06150=1040.411,116.135,407.576,169.955,39.073,157.359
C06151=1040.417,116.384,407.556,169.957,39.074,157.360
C06152=1040.423,116.633,407.535,169.959,39.075,157.360
C06153=1040.429,116.882,407.514,169.962,39.075,157.360
C06154=1040.435,117.131,407.494,169.964,39.076,157.360
C06155=1040.441,117.380,407.474,169.965,39.077,157.360
C06156=1040.447,117.629,407.454,169.967,39.077,157.361
C06157=1040.453,117.879,407.433,169.969,39.078,157.361
C06158=1040.459,118.128,407.413,169.971,39.078,157.361
C06159=1040.466,118.377,407.393,169.974,39.080,157.361
C06160=1040.471,118.626,407.371,169.976,39.080,157.361
C06161=1040.478,118.875,407.351,169.978,39.081,157.362
C06162=1040.484,119.124,407.331,169.980,39.082,157.362
C06163=1040.490,119.373,407.311,169.982,39.082,157.362
C06164=1040.496,119.623,407.290,169.984,39.083,157.362
C06165=1040.502,119.871,407.270,169.987,39.084,157.362
C06166=1040.509,120.120,407.249,169.989,39.084,157.363
C06167=1040.514,120.369,407.229,169.990,39.085,157.363
C06168=1040.521,120.619,407.208,169.992,39.085,157.363
C06169=1040.527,120.867,407.188,169.994,39.086,157.363
C06170=1040.533,121.117,407.167,169.996,39.087,157.363
C06171=1040.539,121.366,407.147,169.999,39.087,157.363
C06172=1040.545,121.615,407.127,170.001,39.088,157.364
C06173=1040.552,121.864,407.106,170.003,39.089,157.364
C06174=1040.557,122.113,407.085,170.005,39.090,157.364
C06175=1040.563,122.362,407.065,170.007,39.090,157.364
C06176=1040.570,122.612,407.045,170.010,39.091,157.365
C06177=1040.576,122.860,407.023,170.012,39.092,157.365
C06178=1040.582,123.110,407.003,170.014,39.092,157.365
C06179=1040.588,123.359,406.983,170.016,39.093,157.365
C06180=1040.594,123.608,406.961,170.018,39.094,157.365
C06181=1040.600,123.857,406.942,170.020,39.094,157.365
C06182=1040.607,124.106,406.921,170.022,39.095,157.366
C06183=1040.612,124.355,406.900,170.025,39.095,157.366
C06184=1040.619,124.604,406.880,170.027,39.096,157.366
C06185=1040.626,124.889,406.856,170.029,39.097,157.366
C06186=1040.634,125.176,406.832,170.031,39.098,157.366
C06187=1040.640,125.462,406.809,170.033,39.099,157.367
C06188=1040.647,125.747,406.785,170.037,39.099,157.367
C06189=1040.654,125.996,406.764,170.039,39.100,157.367
C06190=1040.660,126.246,406.743,170.041,39.101,157.367
C06191=1040.666,126.495,406.723,170.043,39.101,157.367
C06192=1040.672,126.744,406.702,170.045,39.102,157.368
C06193=1040.678,126.993,406.682,170.048,39.103,157.368
C06194=1040.685,127.241,406.661,170.049,39.103,157.368
C06195=1040.690,127.491,406.640,170.051,39.104,157.368
C06196=1040.697,127.739,406.619,170.053,39.104,157.368
C06197=1040.704,127.989,406.599,170.055,39.105,157.369
C06198=1040.710,128.237,406.578,170.057,39.106,157.369
C06199=1040.716,128.487,406.557,170.059,39.106,157.369
C06200=1040.723,128.736,406.536,170.062,39.107,157.369
C06201=1040.728,128.985,406.516,170.064,39.108,157.369
C06202=1040.735,129.234,406.495,170.066,39.108,157.370
C06203=1040.741,129.483,406.475,170.068,39.109,157.370
C06204=1040.747,129.732,406.453,170.070,39.109,157.370
C06205=1040.754,129.981,406.433,170.073,39.111,157.370
C06206=1040.760,130.230,406.412,170.075,39.111,157.370
C06207=1040.766,130.479,406.391,170.077,39.112,157.370
C06208=1040.773,130.728,406.370,170.079,39.112,157.371
C06209=1040.779,130.977,406.350,170.081,39.113,157.371
C06210=1040.785,131.226,406.328,170.083,39.114,157.371
C06211=1040.791,131.476,406.307,170.085,39.114,157.371
C06212=1040.797,131.724,406.287,170.088,39.115,157.372
C06213=1040.803,131.974,406.265,170.090,39.116,157.372
C06214=1040.809,132.223,406.244,170.092,39.117,157.372
C06215=1040.816,132.472,406.224,170.094,39.117,157.372
C06216=1040.822,132.721,406.202,170.096,39.118,157.372
C06217=1040.828,132.970,406.180,170.099,39.119,157.373
C06218=1040.834,133.219,406.160,170.101,39.120,157.373
C06219=1040.840,133.468,406.139,170.103,39.121,157.373
C06220=1040.846,133.717,406.117,170.105,39.121,157.373
C06221=1040.852,133.966,406.097,170.107,39.122,157.373
C06222=1040.858,134.215,406.076,170.110,39.123,157.374
C06223=1040.864,134.464,406.054,170.112,39.123,157.374
C06224=1040.871,134.713,406.033,170.114,39.124,157.374
C06225=1040.877,134.962,406.012,170.116,39.125,157.374
C06226=1040.883,135.212,405.991,170.118,39.125,157.374
C06227=1040.889,135.460,405.970,170.121,39.126,157.375
C06228=1040.895,135.709,405.948,170.123,39.127,157.375
C06229=1040.902,135.958,405.927,170.125,39.127,157.375
C06230=1040.908,136.207,405.907,170.127,39.129,157.375
C06231=1040.914,136.456,405.885,170.129,39.129,157.375
C06232=1040.920,136.706,405.864,170.132,39.130,157.376
C06233=1040.926,136.954,405.843,170.134,39.131,157.376
C06234=1040.932,137.203,405.821,170.136,39.131,157.376
C06235=1040.938,137.452,405.800,170.138,39.132,157.376
C06236=1040.944,137.702,405.779,170.140,39.133,157.376
C06237=1040.951,137.950,405.758,170.142,39.134,157.377
C06238=1040.957,138.199,405.736,170.145,39.134,157.377
C06239=1040.963,138.449,405.715,170.147,39.136,157.377
C06240=1040.969,138.698,405.693,170.149,39.136,157.377
C06241=1040.975,138.946,405.672,170.151,39.136,157.378
C06242=1040.982,139.195,405.651,170.154,39.138,157.378
C06243=1040.988,139.444,405.629,170.157,39.138,157.378
C06244=1040.994,139.694,405.607,170.159,39.139,157.378
C06245=1040.999,139.942,405.586,170.161,39.140,157.378
C06246=1041.006,140.191,405.565,170.163,39.141,157.379
C06247=1041.012,140.440,405.543,170.165,39.141,157.379
C06248=1041.018,140.690,405.521,170.168,39.142,157.379
C06249=1041.025,140.975,405.498,170.170,39.143,157.379
C06250=1041.032,141.261,405.472,170.172,39.144,157.380
C06251=1041.038,141.547,405.448,170.175,39.145,157.380
C06252=1041.046,141.832,405.423,170.178,39.146,157.380
C06253=1041.052,142.081,405.402,170.180,39.147,157.380
C06254=1041.058,142.330,405.380,170.182,39.148,157.381
C06255=1041.064,142.579,405.359,170.184,39.148,157.381
C06256=1041.070,142.828,405.337,170.186,39.149,157.381
C06257=1041.077,143.077,405.316,170.189,39.150,157.381
C06258=1041.082,143.326,405.294,170.191,39.151,157.382
C06259=1041.089,143.574,405.272,170.193,39.151,157.382
C06260=1041.095,143.824,405.250,170.195,39.153,157.382
C06261=1041.101,144.073,405.229,170.197,39.153,157.382
C06262=1041.107,144.322,405.207,170.200,39.154,157.382
C06263=1041.113,144.571,405.186,170.202,39.155,157.383
C06264=1041.119,144.820,405.164,170.204,39.156,157.383
C06265=1041.125,145.069,405.142,170.206,39.156,157.383
C06266=1041.131,145.318,405.121,170.209,39.157,157.383
C06267=1041.138,145.567,405.098,170.212,39.158,157.384
C06268=1041.144,145.816,405.077,170.214,39.158,157.384
C06269=1041.151,146.065,405.056,170.216,39.159,157.384
C06270=1041.156,146.313,405.035,170.218,39.160,157.384
C06271=1041.162,146.563,405.013,170.220,39.161,157.384
C06272=1041.169,146.811,404.991,170.223,39.161,157.385
C06273=1041.175,147.060,404.969,170.225,39.163,157.385
C06274=1041.181,147.310,404.947,170.227,39.164,157.385
C06275=1041.187,147.559,404.925,170.229,39.164,157.385
C06276=1041.193,147.808,404.903,170.231,39.165,157.386
C06277=1041.199,148.057,404.881,170.234,39.166,157.386
C06278=1041.205,148.305,404.860,170.236,39.167,157.386
C06279=1041.211,148.555,404.838,170.238,39.167,157.386
C06280=1041.217,148.803,404.816,170.240,39.169,157.386
C06281=1041.224,149.052,404.794,170.244,39.170,157.387
C06282=1041.230,149.302,404.773,170.246,39.170,157.387
C06283=1041.235,149.551,404.750,170.248,39.171,157.387
C06284=1041.242,149.800,404.728,170.250,39.172,157.387
C06285=1041.248,150.049,404.706,170.252,39.173,157.388
C06286=1041.254,150.298,404.684,170.255,39.174,157.388
C06287=1041.260,150.546,404.663,170.257,39.174,157.388
C06288=1041.266,150.795,404.640,170.259,39.175,157.388
C06289=1041.272,151.044,404.618,170.261,39.176,157.389
C06290=1041.278,151.293,404.596,170.263,39.177,157.389
C06291=1041.284,151.542,404.574,170.266,39.178,157.389
C06292=1041.291,151.791,404.552,170.268,39.179,157.389
C06293=1041.296,152.040,404.530,170.271,39.180,157.390
C06294=1041.302,152.289,404.508,170.273,39.180,157.390
C06295=1041.309,152.538,404.486,170.276,39.181,157.390
C06296=1041.315,152.787,404.464,170.278,39.182,157.390
C06297=1041.322,153.036,404.442,170.280,39.183,157.391
C06298=1041.327,153.285,404.419,170.282,39.184,157.391
C06299=1041.333,153.534,404.397,170.284,39.185,157.391
C06300=1041.340,153.783,404.375,170.287,39.186,157.391
C06301=1041.346,154.031,404.353,170.289,39.187,157.392
C06302=1041.351,154.281,404.331,170.291,39.187,157.392
C06303=1041.358,154.530,404.308,170.294,39.188,157.392
C06304=1041.364,154.779,404.287,170.297,39.189,157.392
C06305=1041.371,155.027,404.264,170.299,39.190,157.392
C06306=1041.375,155.276,404.243,170.301,39.191,157.393
C06307=1041.382,155.525,404.220,170.303,39.192,157.393
C06308=1041.388,155.774,404.197,170.305,39.193,157.393
C06309=1041.394,156.023,404.176,170.308,39.194,157.393
C06310=1041.400,156.271,404.153,170.310,39.195,157.394
C06311=1041.406,156.520,404.130,170.312,39.196,157.394
C06312=1041.412,156.770,404.109,170.315,39.196,157.394
C06313=1041.420,157.055,404.083,170.318,39.197,157.395
C06314=1041.427,157.341,404.057,170.320,39.199,157.395
C06315=1041.433,157.626,404.032,170.323,39.200,157.395
C06316=1041.440,157.911,404.006,170.325,39.201,157.395
C06317=1041.447,158.160,403.983,170.329,39.202,157.396
C06318=1041.453,158.409,403.962,170.331,39.202,157.396
C06319=1041.458,158.658,403.939,170.333,39.203,157.396
C06320=1041.465,158.906,403.916,170.335,39.204,157.396
C06321=1041.471,159.156,403.895,170.337,39.205,157.397
C06322=1041.477,159.404,403.872,170.340,39.206,157.397
C06323=1041.483,159.653,403.850,170.342,39.207,157.397
C06324=1041.489,159.902,403.827,170.345,39.208,157.397
C06325=1041.496,160.152,403.805,170.347,39.209,157.398
C06326=1041.502,160.401,403.782,170.350,39.210,157.398
C06327=1041.508,160.649,403.759,170.352,39.211,157.398
C06328=1041.514,160.898,403.736,170.354,39.212,157.399
C06329=1041.519,161.147,403.713,170.356,39.213,157.399
C06330=1041.525,161.396,403.690,170.359,39.214,157.399
C06331=1041.531,161.645,403.667,170.361,39.215,157.399
C06332=1041.537,161.893,403.645,170.364,39.216,157.400
C06333=1041.543,162.142,403.622,170.366,39.217,157.400
C06334=1041.549,162.392,403.600,170.369,39.218,157.400
C06335=1041.554,162.641,403.577,170.371,39.219,157.400
C06336=1041.561,162.889,403.555,170.373,39.220,157.401
C06337=1041.566,163.138,403.532,170.376,39.221,157.401
C06338=1041.572,163.387,403.509,170.378,39.222,157.401
C06339=1041.578,163.636,403.486,170.380,39.223,157.402
C06340=1041.584,163.885,403.463,170.383,39.225,157.402
C06341=1041.590,164.134,403.441,170.386,39.226,157.402
C06342=1041.596,164.382,403.418,170.388,39.227,157.403
C06343=1041.602,164.631,403.395,170.390,39.228,157.403
C06344=1041.607,164.880,403.372,170.392,39.228,157.403
C06345=1041.613,165.129,403.349,170.395,39.229,157.403
C06346=1041.620,165.378,403.326,170.398,39.230,157.404
C06347=1041.626,165.627,403.302,170.400,39.232,157.404
C06348=1041.632,165.876,403.279,170.402,39.233,157.404
C06349=1041.638,166.125,403.256,170.405,39.234,157.404
C06350=1041.643,166.373,403.234,170.407,39.235,157.405
C06351=1041.650,166.622,403.211,170.409,39.236,157.405
C06352=1041.656,166.871,403.188,170.412,39.237,157.405
C06353=1041.661,167.120,403.165,170.415,39.238,157.406
C06354=1041.668,167.369,403.142,170.417,39.239,157.406
C06355=1041.673,167.618,403.119,170.419,39.240,157.406
C06356=1041.679,167.867,403.096,170.422,39.241,157.406
C06357=1041.686,168.115,403.073,170.424,39.243,157.407
C06358=1041.692,168.364,403.050,170.427,39.243,157.407
C06359=1041.697,168.613,403.027,170.429,39.244,157.407
C06360=1041.704,168.863,403.004,170.431,39.245,157.408
C06361=1041.710,169.104,402.982,170.434,39.246,157.408
C06362=1041.715,169.347,402.959,170.436,39.247,157.408
C06363=1041.721,169.590,402.936,170.438,39.248,157.408
C06364=1041.727,169.832,402.914,170.442,39.250,157.409
C06365=1041.733,170.074,402.891,170.444,39.251,157.409
C06366=1041.739,170.317,402.870,170.446,39.252,157.409
C06367=1041.745,170.560,402.847,170.448,39.253,157.410
C06368=1041.751,170.803,402.824,170.451,39.253,157.410
C06369=1041.757,171.051,402.801,170.453,39.254,157.410
C06370=1041.763,171.299,402.778,170.456,39.255,157.410
C06371=1041.769,171.548,402.755,170.458,39.257,157.411
C06372=1041.775,171.798,402.731,170.461,39.258,157.411
C06373=1041.781,172.047,402.708,170.463,39.259,157.411
C06374=1041.787,172.295,402.685,170.466,39.260,157.412
C06375=1041.793,172.544,402.662,170.468,39.261,157.412
C06376=1041.800,172.793,402.639,170.471,39.262,157.412
C06377=1041.807,173.090,402.611,170.474,39.263,157.412
C06378=1041.814,173.388,402.584,170.477,39.265,157.413
C06379=1041.821,173.686,402.555,170.480,39.266,157.413
C06380=1041.828,173.983,402.527,170.483,39.267,157.413
C06381=1041.835,174.232,402.505,170.485,39.268,157.414
C06382=1041.841,174.481,402.481,170.487,39.269,157.414
C06383=1041.847,174.730,402.458,170.491,39.270,157.414
C06384=1041.853,174.978,402.434,170.493,39.271,157.415
C06385=1041.860,175.228,402.411,170.495,39.272,157.415
C06386=1041.865,175.476,402.388,170.499,39.273,157.415
C06387=1041.871,175.725,402.365,170.501,39.274,157.416
C06388=1041.878,175.974,402.341,170.503,39.275,157.416
C06389=1041.884,176.222,402.318,170.505,39.277,157.416
C06390=1041.890,176.471,402.295,170.509,39.278,157.416
C06391=1041.897,176.720,402.271,170.511,39.279,157.417
C06392=1041.902,176.969,402.248,170.513,39.280,157.417
C06393=1041.909,177.218,402.224,170.517,39.281,157.417
C06394=1041.915,177.467,402.201,170.519,39.282,157.418
C06395=1041.921,177.715,402.178,170.521,39.283,157.418
C06396=1041.927,177.965,402.154,170.523,39.284,157.418
C06397=1041.933,178.213,402.131,170.527,39.285,157.418
C06398=1041.940,178.462,402.108,170.529,39.286,157.419
C06399=1041.946,178.711,402.084,170.531,39.287,157.419
C06400=1041.952,178.960,402.061,170.534,39.288,157.419
C06401=1041.959,179.209,402.037,170.537,39.289,157.420
C06402=1041.964,179.457,402.014,170.539,39.291,157.420
C06403=1041.971,179.706,401.990,170.542,39.292,157.420
C06404=1041.977,179.955,401.967,170.545,39.293,157.421
C06405=1041.983,180.204,401.943,170.547,39.294,157.421
C06406=1041.990,180.453,401.920,170.550,39.295,157.421
C06407=1041.996,180.702,401.896,170.552,39.296,157.421
C06408=1042.002,180.950,401.873,170.555,39.297,157.422
C06409=1042.009,181.199,401.849,170.558,39.298,157.422
C06410=1042.015,181.448,401.826,170.560,39.299,157.422
C06411=1042.022,181.697,401.802,170.562,39.300,157.423
C06412=1042.028,181.945,401.779,170.566,39.301,157.423
C06413=1042.034,182.195,401.755,170.568,39.302,157.423
C06414=1042.040,182.443,401.732,170.570,39.303,157.424
C06415=1042.047,182.692,401.708,170.574,39.304,157.424
C06416=1042.053,182.940,401.684,170.576,39.306,157.424
C06417=1042.059,183.190,401.661,170.579,39.307,157.424
C06418=1042.065,183.438,401.637,170.581,39.308,157.425
C06419=1042.072,183.687,401.613,170.584,39.309,157.425
C06420=1042.078,183.935,401.589,170.587,39.310,157.425
C06421=1042.084,184.185,401.565,170.589,39.311,157.426
C06422=1042.090,184.433,401.541,170.592,39.313,157.426
C06423=1042.095,184.682,401.518,170.595,39.314,157.427
C06424=1042.101,184.931,401.493,170.597,39.315,157.427
C06425=1042.107,185.180,401.469,170.600,39.316,157.427
C06426=1042.113,185.429,401.445,170.603,39.318,157.428
C06427=1042.119,185.677,401.421,170.605,39.319,157.428
C06428=1042.125,185.926,401.397,170.608,39.320,157.428
C06429=1042.130,186.175,401.373,170.611,39.322,157.429
C06430=1042.137,186.424,401.349,170.613,39.323,157.429
C06431=1042.142,186.673,401.324,170.615,39.324,157.429
C06432=1042.149,186.922,401.300,170.619,39.326,157.430
C06433=1042.154,187.170,401.276,170.621,39.327,157.430
C06434=1042.161,187.419,401.252,170.624,39.329,157.430
C06435=1042.166,187.668,401.228,170.627,39.330,157.431
C06436=1042.173,187.917,401.204,170.629,39.331,157.431
C06437=1042.178,188.165,401.180,170.632,39.332,157.431
C06438=1042.185,188.414,401.155,170.635,39.333,157.432
C06439=1042.190,188.662,401.131,170.637,39.334,157.432
C06440=1042.197,188.911,401.106,170.639,39.336,157.432
C06441=1042.204,189.195,401.080,170.643,39.338,157.433
C06442=1042.211,189.480,401.051,170.646,39.339,157.433
C06443=1042.217,189.765,401.023,170.650,39.340,157.434
C06444=1042.225,190.049,400.995,170.652,39.342,157.434
C06445=1042.231,190.297,400.972,170.655,39.343,157.434
C06446=1042.237,190.546,400.947,170.658,39.344,157.435
C06447=1042.243,190.795,400.923,170.660,39.346,157.435
C06448=1042.248,191.044,400.899,170.663,39.347,157.435
C06449=1042.255,191.292,400.874,170.666,39.349,157.436
C06450=1042.261,191.541,400.850,170.669,39.350,157.436
C06451=1042.267,191.790,400.825,170.671,39.351,157.436
C06452=1042.273,192.039,400.802,170.674,39.353,157.437
C06453=1042.279,192.288,400.777,170.677,39.354,157.437
C06454=1042.285,192.536,400.752,170.679,39.355,157.437
C06455=1042.291,192.785,400.728,170.683,39.356,157.438
C06456=1042.297,193.034,400.704,170.685,39.358,157.438
C06457=1042.304,193.282,400.679,170.687,39.359,157.439
C06458=1042.310,193.531,400.655,170.691,39.360,157.439
C06459=1042.316,193.780,400.630,170.693,39.362,157.439
C06460=1042.322,194.029,400.606,170.696,39.363,157.440
C06461=1042.328,194.277,400.581,170.699,39.365,157.440
C06462=1042.334,194.526,400.557,170.702,39.366,157.440
C06463=1042.340,194.775,400.533,170.704,39.367,157.441
C06464=1042.346,195.023,400.508,170.708,39.368,157.441
C06465=1042.353,195.272,400.484,170.710,39.370,157.441
C06466=1042.359,195.521,400.458,170.712,39.371,157.442
C06467=1042.365,195.770,400.434,170.716,39.372,157.442
C06468=1042.371,196.018,400.410,170.718,39.374,157.443
C06469=1042.378,196.267,400.385,170.721,39.375,157.443
C06470=1042.384,196.516,400.361,170.724,39.376,157.443
C06471=1042.391,196.764,400.336,170.727,39.377,157.444
C06472=1042.396,197.013,400.312,170.729,39.379,157.444
C06473=1042.402,197.262,400.287,170.733,39.380,157.444
C06474=1042.409,197.511,400.262,170.735,39.382,157.445
C06475=1042.415,197.760,400.238,170.738,39.383,157.445
C06476=1042.421,198.008,400.213,170.741,39.385,157.445
C06477=1042.427,198.257,400.189,170.744,39.386,157.446
C06478=1042.434,198.505,400.164,170.746,39.387,157.446
C06479=1042.440,198.755,400.139,170.750,39.388,157.447
C06480=1042.446,199.003,400.114,170.752,39.390,157.447
C06481=1042.452,199.251,400.090,170.755,39.391,157.447
C06482=1042.458,199.500,400.065,170.758,39.393,157.448
C06483=1042.465,199.748,400.040,170.761,39.394,157.448
C06484=1042.471,199.998,400.016,170.764,39.395,157.448
C06485=1042.477,200.246,399.990,170.767,39.396,157.449
C06486=1042.484,200.495,399.966,170.769,39.398,157.449
C06487=1042.489,200.743,399.941,170.773,39.399,157.449
C06488=1042.496,200.992,399.917,170.775,39.401,157.450
C06489=1042.502,201.241,399.892,170.778,39.403,157.450
C06490=1042.508,201.490,399.867,170.781,39.404,157.451
C06491=1042.514,201.739,399.842,170.784,39.405,157.451
C06492=1042.521,201.988,399.817,170.786,39.407,157.451
C06493=1042.526,202.236,399.792,170.790,39.408,157.452
C06494=1042.532,202.484,399.766,170.792,39.410,157.452
C06495=1042.538,202.734,399.742,170.796,39.411,157.453
C06496=1042.545,202.982,399.717,170.798,39.413,157.453
C06497=1042.551,203.231,399.692,170.801,39.414,157.453
C06498=1042.558,203.479,399.666,170.804,39.416,157.454
C06499=1042.563,203.727,399.641,170.807,39.417,157.454
C06500=1042.569,203.977,399.617,170.810,39.419,157.455
C06501=1042.575,204.225,399.591,170.813,39.420,157.455
C06502=1042.582,204.474,399.566,170.815,39.422,157.455
C06503=1042.588,204.723,399.541,170.819,39.423,157.456
C06504=1042.594,204.971,399.515,170.822,39.425,157.456
C06505=1042.620,206.023,399.409,171.095,39.527,157.487
C06506=1042.628,206.315,399.378,171.097,39.530,157.487
C06507=1042.636,206.607,399.347,171.100,39.533,157.488
C06508=1042.643,206.899,399.316,171.102,39.535,157.488
C06509=1042.651,207.192,399.285,171.105,39.538,157.489
C06510=1042.658,207.440,399.259,171.107,39.540,157.490
C06511=1042.665,207.688,399.232,171.109,39.542,157.490
C06512=1042.672,207.937,399.206,171.111,39.544,157.491
C06513=1042.678,208.186,399.179,171.114,39.546,157.491
C06514=1042.685,208.434,399.153,171.115,39.549,157.492
C06515=1042.692,208.683,399.127,171.118,39.551,157.492
C06516=1042.697,208.931,399.100,171.120,39.554,157.493
C06517=1042.705,209.180,399.074,171.122,39.556,157.494
C06518=1042.711,209.428,399.047,171.125,39.558,157.494
C06519=1042.717,209.677,399.020,171.126,39.560,157.495
C06520=1042.724,209.925,398.994,171.129,39.563,157.495
C06521=1042.731,210.174,398.968,171.131,39.565,157.496
C06522=1042.737,210.423,398.941,171.133,39.567,157.496
C06523=1042.744,210.671,398.915,171.135,39.569,157.497
C06524=1042.751,210.920,398.887,171.138,39.571,157.497
C06525=1042.757,211.168,398.861,171.139,39.574,157.498
C06526=1042.764,211.416,398.835,171.142,39.576,157.498
C06527=1042.771,211.666,398.808,171.144,39.578,157.499
C06528=1042.777,211.914,398.782,171.146,39.581,157.500
C06529=1042.784,212.163,398.755,171.149,39.583,157.500
C06530=1042.790,212.410,398.728,171.150,39.585,157.501
C06531=1042.797,212.659,398.701,171.153,39.588,157.501
C06532=1042.804,212.908,398.674,171.155,39.590,157.502
C06533=1042.810,213.156,398.648,171.157,39.592,157.502
C06534=1042.817,213.404,398.621,171.159,39.594,157.503
C06535=1042.823,213.653,398.594,171.162,39.596,157.503
C06536=1042.829,213.902,398.567,171.163,39.599,157.504
C06537=1042.836,214.151,398.541,171.166,39.601,157.504
C06538=1042.842,214.398,398.513,171.169,39.603,157.505
C06539=1042.849,214.647,398.487,171.170,39.606,157.506
C06540=1042.855,214.895,398.460,171.173,39.608,157.506
C06541=1042.863,215.144,398.433,171.175,39.610,157.507
C06542=1042.869,215.393,398.406,171.177,39.613,157.507
C06543=1042.875,215.641,398.379,171.179,39.615,157.508
C06544=1042.882,215.889,398.352,171.182,39.617,157.508
C06545=1042.889,216.138,398.325,171.184,39.619,157.509
C06546=1042.895,216.386,398.299,171.186,39.621,157.509
C06547=1042.902,216.635,398.271,171.188,39.624,157.510
C06548=1042.909,216.883,398.245,171.191,39.626,157.511
C06549=1042.915,217.131,398.218,171.193,39.628,157.511
C06550=1042.921,217.380,398.191,171.195,39.630,157.512
C06551=1042.928,217.629,398.164,171.198,39.633,157.512
C06552=1042.935,217.877,398.136,171.200,39.635,157.513
C06553=1042.942,218.125,398.110,171.202,39.637,157.513
C06554=1042.948,218.374,398.083,171.204,39.639,157.514
C06555=1042.955,218.623,398.056,171.207,39.641,157.514
C06556=1042.962,218.871,398.029,171.209,39.644,157.515
C06557=1042.968,219.119,398.002,171.211,39.646,157.515
C06558=1042.975,219.368,397.975,171.214,39.648,157.516
C06559=1042.982,219.617,397.948,171.216,39.651,157.517
C06560=1042.989,219.865,397.921,171.219,39.652,157.517
C06561=1042.995,220.113,397.894,171.220,39.655,157.518
C06562=1043.003,220.411,397.861,171.223,39.658,157.518
C06563=1043.011,220.709,397.828,171.226,39.660,157.519
C06564=1043.019,221.006,397.796,171.229,39.663,157.520
C06565=1043.026,221.305,397.763,171.232,39.666,157.520
C06566=1043.033,221.554,397.736,171.233,39.668,157.521
C06567=1043.039,221.801,397.708,171.236,39.670,157.521
C06568=1043.046,222.050,397.682,171.239,39.672,157.522
C06569=1043.053,222.298,397.654,171.241,39.675,157.523
C06570=1043.059,222.547,397.626,171.243,39.677,157.523
C06571=1043.065,222.795,397.600,171.245,39.679,157.524
C06572=1043.072,223.044,397.572,171.248,39.682,157.524
C06573=1043.078,223.292,397.544,171.250,39.684,157.525
C06574=1043.085,223.541,397.517,171.253,39.686,157.525
C06575=1043.092,223.789,397.490,171.254,39.688,157.526
C06576=1043.098,224.037,397.463,171.257,39.690,157.526
C06577=1043.105,224.286,397.435,171.259,39.693,157.527
C06578=1043.112,224.534,397.407,171.262,39.695,157.528
C06579=1043.118,224.783,397.380,171.265,39.697,157.528
C06580=1043.125,225.032,397.353,171.266,39.699,157.529
C06581=1043.131,225.279,397.325,171.269,39.702,157.529
C06582=1043.138,225.527,397.298,171.271,39.704,157.530
C06583=1043.145,225.776,397.271,171.274,39.706,157.530
C06584=1043.151,226.025,397.243,171.276,39.708,157.531
C06585=1043.158,226.273,397.216,171.278,39.710,157.531
C06586=1043.165,226.522,397.188,171.280,39.713,157.532
C06587=1043.171,226.770,397.160,171.283,39.715,157.533
C06588=1043.177,227.018,397.133,171.286,39.717,157.533
C06589=1043.184,227.267,397.106,171.288,39.719,157.534
C06590=1043.190,227.515,397.078,171.291,39.722,157.534
C06591=1043.198,227.764,397.051,171.292,39.724,157.535
C06592=1043.205,228.012,397.023,171.295,39.726,157.535
C06593=1043.211,228.260,396.995,171.297,39.728,157.536
C06594=1043.218,228.509,396.968,171.300,39.730,157.536
C06595=1043.225,228.757,396.940,171.303,39.733,157.537
C06596=1043.231,229.006,396.912,171.305,39.735,157.538
C06597=1043.237,229.254,396.885,171.308,39.737,157.538
C06598=1043.244,229.502,396.857,171.309,39.739,157.539
C06599=1043.250,229.751,396.829,171.312,39.742,157.539
C06600=1043.257,229.999,396.801,171.314,39.744,157.540
C06601=1043.263,230.248,396.773,171.317,39.746,157.540
C06602=1043.270,230.496,396.746,171.320,39.749,157.541
C06603=1043.277,230.744,396.718,171.322,39.751,157.542
C06604=1043.283,230.993,396.690,171.325,39.753,157.542
C06605=1043.290,231.241,396.662,171.326,39.755,157.543
C06606=1043.297,231.490,396.635,171.329,39.757,157.543
C06607=1043.303,231.738,396.607,171.331,39.759,157.544
C06608=1043.309,231.986,396.579,171.334,39.762,157.544
C06609=1043.315,232.235,396.551,171.336,39.764,157.545
C06610=1043.322,232.483,396.523,171.339,39.766,157.545
C06611=1043.329,232.731,396.495,171.342,39.768,157.546
C06612=1043.335,232.980,396.467,171.344,39.771,157.547
C06613=1043.342,233.228,396.439,171.347,39.773,157.547
C06614=1043.348,233.477,396.411,171.348,39.775,157.548
C06615=1043.355,233.725,396.384,171.351,39.778,157.548
C06616=1043.361,233.973,396.355,171.353,39.780,157.549
C06617=1043.368,234.222,396.327,171.356,39.782,157.549
C06618=1043.376,234.511,396.294,171.359,39.785,157.550
C06619=1043.384,234.803,396.261,171.362,39.787,157.551
C06620=1043.392,235.093,396.229,171.365,39.790,157.551
C06621=1043.399,235.383,396.196,171.368,39.793,157.552
C06622=1043.406,235.631,396.168,171.370,39.795,157.553
C06623=1043.412,235.880,396.139,171.373,39.797,157.553
C06624=1043.418,236.128,396.112,171.375,39.799,157.554
C06625=1043.425,236.376,396.083,171.378,39.801,157.554
C06626=1043.432,236.625,396.055,171.381,39.804,157.555
C06627=1043.438,236.873,396.027,171.383,39.806,157.556
C06628=1043.445,237.121,395.999,171.386,39.808,157.556
C06629=1043.451,237.370,395.971,171.388,39.810,157.557
C06630=1043.458,237.618,395.943,171.391,39.813,157.557
C06631=1043.464,237.866,395.914,171.394,39.815,157.558
C06632=1043.472,238.115,395.886,171.396,39.817,157.558
C06633=1043.479,238.363,395.858,171.399,39.820,157.559
C06634=1043.485,238.612,395.829,171.401,39.822,157.560
C06635=1043.491,238.860,395.802,171.403,39.824,157.560
C06636=1043.498,239.108,395.773,171.405,39.826,157.561
C06637=1043.504,239.357,395.745,171.408,39.829,157.561
C06638=1043.511,239.605,395.716,171.411,39.831,157.562
C06639=1043.517,239.853,395.688,171.413,39.833,157.562
C06640=1043.524,240.101,395.660,171.416,39.835,157.563
C06641=1043.531,240.350,395.632,171.418,39.837,157.563
C06642=1043.537,240.598,395.603,171.421,39.839,157.564
C06643=1043.544,240.847,395.575,171.423,39.842,157.565
C06644=1043.551,241.095,395.546,171.426,39.844,157.565
C06645=1043.557,241.344,395.518,171.429,39.846,157.566
C06646=1043.564,241.591,395.489,171.431,39.848,157.566
C06647=1043.571,241.839,395.460,171.434,39.851,157.567
C06648=1043.576,242.088,395.432,171.436,39.853,157.568
C06649=1043.583,242.336,395.404,171.439,39.855,157.568
C06650=1043.589,242.585,395.375,171.441,39.857,157.569
C06651=1043.596,242.833,395.347,171.444,39.860,157.569
C06652=1043.603,243.081,395.318,171.447,39.862,157.570
C06653=1043.609,243.330,395.288,171.449,39.864,157.570
C06654=1043.616,243.578,395.261,171.452,39.866,157.571
C06655=1043.622,243.826,395.232,171.454,39.869,157.572
C06656=1043.629,244.074,395.203,171.457,39.872,157.572
C06657=1043.635,244.323,395.175,171.461,39.874,157.573
C06658=1043.642,244.571,395.146,171.463,39.876,157.573
C06659=1043.649,244.819,395.117,171.466,39.878,157.574
C06660=1043.655,245.068,395.088,171.469,39.881,157.575
C06661=1043.662,245.316,395.060,171.471,39.883,157.575
C06662=1043.668,245.564,395.031,171.474,39.885,157.576
C06663=1043.675,245.812,395.002,171.476,39.887,157.576
C06664=1043.681,246.060,394.973,171.479,39.890,157.577
C06665=1043.687,246.309,394.944,171.481,39.892,157.578
C06666=1043.693,246.557,394.915,171.484,39.894,157.578
C06667=1043.701,246.805,394.886,171.487,39.896,157.579
C06668=1043.707,247.053,394.857,171.489,39.899,157.579
C06669=1043.713,247.302,394.829,171.492,39.901,157.580
C06670=1043.719,247.550,394.800,171.495,39.904,157.581
C06671=1043.726,247.798,394.771,171.497,39.906,157.581
C06672=1043.732,248.046,394.742,171.500,39.908,157.582
C06673=1043.739,248.295,394.712,171.502,39.910,157.582
C06674=1043.746,248.579,394.679,171.506,39.913,157.583
C06675=1043.754,248.864,394.646,171.509,39.915,157.584
C06676=1043.761,249.148,394.613,171.511,39.918,157.584
C06677=1043.768,249.433,394.580,171.515,39.921,157.585
C06678=1043.775,249.682,394.551,171.518,39.923,157.586
C06679=1043.782,249.930,394.522,171.520,39.926,157.586
C06680=1043.788,250.177,394.492,171.523,39.928,157.587
C06681=1043.794,250.425,394.463,171.526,39.930,157.587
C06682=1043.801,250.674,394.433,171.528,39.932,157.588
C06683=1043.807,250.922,394.404,171.531,39.935,157.589
C06684=1043.814,251.170,394.376,171.533,39.937,157.589
C06685=1043.821,251.418,394.347,171.536,39.940,157.590
C06686=1043.827,251.667,394.317,171.540,39.942,157.590
C06687=1043.834,251.915,394.288,171.542,39.944,157.591
C06688=1043.840,252.164,394.259,171.545,39.946,157.592
C06689=1043.847,252.412,394.229,171.547,39.949,157.592
C06690=1043.853,252.660,394.200,171.550,39.951,157.593
C06691=1043.860,252.908,394.171,171.553,39.953,157.593
C06692=1043.867,253.157,394.142,171.555,39.955,157.594
C06693=1043.873,253.405,394.113,171.559,39.958,157.595
C06694=1043.880,253.653,394.084,171.562,39.960,157.595
C06695=1043.887,253.901,394.054,171.564,39.963,157.596
C06696=1043.893,254.149,394.025,171.567,39.965,157.596
C06697=1043.899,254.397,393.996,171.569,39.967,157.597
C06698=1043.906,254.646,393.967,171.572,39.969,157.598
C06699=1043.913,254.894,393.937,171.575,39.971,157.598
C06700=1043.919,255.142,393.908,171.578,39.974,157.599
C06701=1043.926,255.391,393.878,171.581,39.976,157.599
C06702=1043.932,255.638,393.849,171.583,39.978,157.600
C06703=1043.939,255.887,393.819,171.586,39.980,157.601
C06704=1043.946,256.135,393.790,171.589,39.983,157.601
C06705=1043.952,256.383,393.760,171.592,39.985,157.602
C06706=1043.960,256.631,393.732,171.595,39.988,157.602
C06707=1043.966,256.879,393.703,171.598,39.990,157.603
C06708=1043.973,257.127,393.672,171.600,39.992,157.604
C06709=1043.979,257.376,393.643,171.603,39.994,157.604
C06710=1043.986,257.624,393.614,171.606,39.996,157.605
C06711=1043.993,257.872,393.584,171.609,39.999,157.605
C06712=1043.999,258.120,393.555,171.612,40.001,157.606
C06713=1044.006,258.368,393.525,171.614,40.003,157.607
C06714=1044.012,258.616,393.496,171.618,40.005,157.607
C06715=1044.020,258.865,393.466,171.620,40.008,157.608
C06716=1044.026,259.113,393.437,171.623,40.010,157.608
C06717=1044.033,259.362,393.408,171.626,40.013,157.609
C06718=1044.039,259.609,393.378,171.629,40.015,157.610
C06719=1044.046,259.858,393.348,171.632,40.017,157.610
C06720=1044.053,260.105,393.319,171.635,40.019,157.611
C06721=1044.060,260.354,393.288,171.637,40.021,157.611
C06722=1044.066,260.602,393.259,171.641,40.024,157.612
C06723=1044.073,260.850,393.229,171.643,40.026,157.613
C06724=1044.079,261.098,393.200,171.646,40.028,157.613
C06725=1044.087,261.346,393.171,171.649,40.030,157.614
C06726=1044.094,261.595,393.141,171.652,40.032,157.614
C06727=1044.101,261.842,393.112,171.655,40.035,157.615
C06728=1044.108,262.091,393.082,171.657,40.037,157.616
C06729=1044.114,262.339,393.052,171.661,40.040,157.616
C06730=1044.121,262.622,393.018,171.664,40.042,157.617
C06731=1044.129,262.905,392.984,171.668,40.045,157.618
C06732=1044.136,263.189,392.950,171.670,40.047,157.618
C06733=1044.144,263.471,392.916,171.674,40.050,157.619
C06734=1044.150,263.720,392.885,171.677,40.052,157.620
C06735=1044.157,263.967,392.855,171.679,40.055,157.620
C06736=1044.164,264.216,392.825,171.683,40.057,157.621
C06737=1044.170,264.463,392.795,171.686,40.060,157.622
C06738=1044.177,264.712,392.765,171.688,40.062,157.622
C06739=1044.184,264.961,392.735,171.692,40.065,157.623
C06740=1044.190,265.208,392.705,171.695,40.067,157.624
C06741=1044.197,265.457,392.675,171.697,40.069,157.624
C06742=1044.203,265.704,392.645,171.700,40.071,157.625
C06743=1044.210,265.953,392.614,171.704,40.074,157.626
C06744=1044.216,266.200,392.585,171.706,40.076,157.626
C06745=1044.223,266.448,392.555,171.709,40.078,157.627
C06746=1044.230,266.697,392.524,171.712,40.081,157.627
C06747=1044.236,266.944,392.494,171.715,40.083,157.628
C06748=1044.243,267.193,392.465,171.718,40.086,157.629
C06749=1044.250,267.442,392.434,171.721,40.088,157.629
C06750=1044.256,267.689,392.404,171.724,40.090,157.630
C06751=1044.263,267.938,392.374,171.727,40.093,157.631
C06752=1044.269,268.185,392.344,171.730,40.095,157.631
C06753=1044.276,268.434,392.313,171.733,40.097,157.632
C06754=1044.283,268.681,392.282,171.736,40.100,157.632
C06755=1044.290,268.929,392.252,171.739,40.102,157.633
C06756=1044.296,269.177,392.222,171.742,40.104,157.634
C06757=1044.303,269.426,392.192,171.745,40.107,157.634
C06758=1044.309,269.673,392.161,171.748,40.109,157.635
C06759=1044.316,269.922,392.131,171.751,40.112,157.636
C06760=1044.323,270.170,392.100,171.754,40.114,157.636
C06761=1044.328,270.418,392.070,171.757,40.116,157.637
C06762=1044.335,270.666,392.040,171.760,40.119,157.638
C06763=1044.342,270.914,392.009,171.764,40.121,157.638
C06764=1044.349,271.162,391.979,171.766,40.124,157.639
C06765=1044.355,271.410,391.948,171.769,40.126,157.639
C06766=1044.362,271.658,391.918,171.773,40.129,157.640
C06767=1044.368,271.906,391.888,171.775,40.131,157.641
C06768=1044.376,272.154,391.857,171.778,40.133,157.641
C06769=1044.382,272.402,391.826,171.782,40.136,157.642
C06770=1044.388,272.650,391.796,171.784,40.138,157.643
C06771=1044.395,272.898,391.765,171.788,40.141,157.643
C06772=1044.402,273.146,391.734,171.791,40.143,157.644
C06773=1044.408,273.395,391.703,171.793,40.145,157.645
C06774=1044.415,273.642,391.673,171.797,40.148,157.645
C06775=1044.421,273.890,391.642,171.800,40.150,157.646
C06776=1044.428,274.139,391.611,171.804,40.153,157.647
C06777=1044.435,274.386,391.581,171.806,40.155,157.647
C06778=1044.441,274.634,391.550,171.810,40.158,157.648
C06779=1044.448,274.882,391.519,171.813,40.160,157.649
C06780=1044.455,275.130,391.489,171.815,40.162,157.649
C06781=1044.461,275.379,391.458,171.819,40.165,157.650
C06782=1044.468,275.626,391.427,171.822,40.167,157.651
C06783=1044.474,275.874,391.396,171.825,40.170,157.651
C06784=1044.481,276.122,391.365,171.828,40.172,157.652
C06785=1044.488,276.371,391.335,171.832,40.175,157.653
C06786=1044.495,276.658,391.298,171.834,40.178,157.653
C06787=1044.504,276.945,391.262,171.838,40.180,157.654
C06788=1044.510,277.233,391.227,171.842,40.183,157.655
C06789=1044.519,277.521,391.191,171.846,40.186,157.656
C06790=1044.525,277.768,391.160,171.849,40.189,157.656
C06791=1044.532,278.016,391.129,171.852,40.191,157.657
C06792=1044.539,278.265,391.099,171.855,40.193,157.658
C06793=1044.545,278.513,391.067,171.859,40.196,157.658
C06794=1044.552,278.760,391.036,171.861,40.198,157.659
C06795=1044.558,279.009,391.005,171.865,40.200,157.660
C06796=1044.565,279.256,390.974,171.868,40.203,157.660
C06797=1044.571,279.504,390.943,171.871,40.205,157.661
C06798=1044.578,279.753,390.912,171.874,40.208,157.662
C06799=1044.584,280.000,390.880,171.878,40.211,157.663
C06800=1044.591,280.248,390.849,171.881,40.213,157.663
C06801=1044.598,280.496,390.818,171.884,40.216,157.664
C06802=1044.605,280.744,390.786,171.887,40.218,157.665
C06803=1044.610,280.992,390.756,171.891,40.221,157.665
C06804=1044.617,281.240,390.724,171.894,40.224,157.666
C06805=1044.624,281.488,390.693,171.897,40.226,157.667
C06806=1044.631,281.736,390.661,171.900,40.228,157.667
C06807=1044.637,281.984,390.630,171.904,40.231,157.668
C06808=1044.644,282.232,390.599,171.906,40.233,157.669
C06809=1044.651,282.479,390.567,171.910,40.236,157.669
C06810=1044.657,282.728,390.536,171.913,40.238,157.670
C06811=1044.664,282.976,390.505,171.917,40.241,157.671
C06812=1044.671,283.224,390.474,171.919,40.243,157.671
C06813=1044.677,283.472,390.442,171.923,40.246,157.672
C06814=1044.684,283.720,390.411,171.926,40.249,157.673
C06815=1044.691,283.967,390.379,171.929,40.251,157.674
C06816=1044.698,284.215,390.348,171.933,40.254,157.674
C06817=1044.704,284.463,390.316,171.936,40.256,157.675
C06818=1044.711,284.711,390.285,171.940,40.258,157.676
C06819=1044.718,284.959,390.254,171.942,40.261,157.676
C06820=1044.724,285.207,390.222,171.946,40.263,157.677
C06821=1044.731,285.455,390.191,171.949,40.266,157.678
C06822=1044.738,285.703,390.159,171.953,40.269,157.678
C06823=1044.745,285.951,390.128,171.956,40.271,157.679
C06824=1044.751,286.199,390.096,171.959,40.274,157.680
C06825=1044.758,286.446,390.064,171.963,40.276,157.681
C06826=1044.765,286.694,390.033,171.965,40.279,157.681
C06827=1044.772,286.942,390.001,171.969,40.281,157.682
C06828=1044.779,287.190,389.970,171.973,40.284,157.683
C06829=1044.785,287.437,389.938,171.976,40.286,157.683
C06830=1044.791,287.686,389.906,171.979,40.289,157.684
C06831=1044.798,287.933,389.874,171.982,40.292,157.685
C06832=1044.805,288.181,389.843,171.986,40.294,157.686
C06833=1044.812,288.429,389.811,171.990,40.296,157.686
C06834=1044.818,288.677,389.779,171.992,40.299,157.687
C06835=1044.825,288.924,389.747,171.996,40.302,157.688
C06836=1044.831,289.172,389.716,171.999,40.305,157.688
C06837=1044.838,289.420,389.684,172.003,40.307,157.689
C06838=1044.845,289.668,389.651,172.006,40.310,157.690
C06839=1044.852,289.916,389.620,172.009,40.312,157.691
C06840=1044.859,290.164,389.588,172.013,40.315,157.691
C06841=1044.865,290.412,389.556,172.017,40.318,157.692
C06842=1044.873,290.711,389.518,172.021,40.320,157.693
C06843=1044.881,291.011,389.479,172.025,40.324,157.694
C06844=1044.889,291.309,389.440,172.028,40.327,157.695
C06845=1044.897,291.609,389.401,172.032,40.330,157.695
C06846=1044.904,291.856,389.369,172.036,40.333,157.696
C06847=1044.911,292.104,389.338,172.040,40.336,157.697
C06848=1044.917,292.352,389.305,172.043,40.338,157.698
C06849=1044.924,292.600,389.274,172.046,40.340,157.698
C06850=1044.931,292.848,389.241,172.050,40.343,157.699
C06851=1044.937,293.096,389.209,172.053,40.346,157.700
C06852=1044.944,293.343,389.177,172.057,40.349,157.701
C06853=1044.951,293.591,389.146,172.061,40.351,157.701
C06854=1044.957,293.839,389.113,172.063,40.354,157.702
C06855=1044.965,294.087,389.081,172.067,40.356,157.703
C06856=1044.971,294.335,389.048,172.071,40.359,157.704
C06857=1044.978,294.582,389.016,172.074,40.362,157.704
C06858=1044.984,294.830,388.984,172.077,40.364,157.705
C06859=1044.991,295.078,388.952,172.081,40.367,157.706
C06860=1044.998,295.326,388.919,172.085,40.370,157.707
C06861=1045.005,295.573,388.887,172.088,40.372,157.707
C06862=1045.011,295.821,388.855,172.092,40.375,157.708
C06863=1045.018,296.069,388.823,172.095,40.378,157.709
C06864=1045.025,296.317,388.789,172.098,40.381,157.710
C06865=1045.031,296.565,388.757,172.102,40.383,157.710
C06866=1045.038,296.812,388.724,172.106,40.386,157.711
C06867=1045.045,297.059,388.692,172.110,40.389,157.712
C06868=1045.051,297.308,388.660,172.113,40.392,157.713
C06869=1045.057,297.556,388.627,172.116,40.395,157.713
C06870=1045.064,297.804,388.594,172.120,40.397,157.714
C06871=1045.070,298.051,388.561,172.123,40.400,157.715
C06872=1045.077,298.298,388.529,172.127,40.403,157.716
C06873=1045.084,298.547,388.496,172.131,40.406,157.717
C06874=1045.090,298.794,388.463,172.134,40.408,157.717
C06875=1045.097,299.042,388.430,172.137,40.412,157.718
C06876=1045.104,299.289,388.398,172.141,40.414,157.719
C06877=1045.110,299.538,388.365,172.145,40.417,157.720
C06878=1045.117,299.785,388.332,172.149,40.420,157.720
C06879=1045.123,300.033,388.300,172.152,40.422,157.721
C06880=1045.130,300.281,388.267,172.155,40.425,157.722
C06881=1045.136,300.529,388.234,172.159,40.428,157.723
C06882=1045.144,300.775,388.201,172.163,40.431,157.724
C06883=1045.150,301.024,388.168,172.166,40.434,157.724
C06884=1045.157,301.271,388.135,172.170,40.436,157.725
C06885=1045.163,301.519,388.102,172.174,40.439,157.726
C06886=1045.170,301.767,388.069,172.177,40.442,157.727
C06887=1045.177,302.014,388.037,172.181,40.445,157.728
C06888=1045.184,302.262,388.003,172.184,40.448,157.728
C06889=1045.190,302.510,387.971,172.188,40.450,157.729
C06890=1045.197,302.757,387.938,172.192,40.453,157.730
C06891=1045.204,303.005,387.905,172.196,40.456,157.731
C06892=1045.210,303.253,387.872,172.200,40.459,157.732
C06893=1045.218,303.500,387.839,172.203,40.462,157.732
C06894=1045.224,303.748,387.806,172.206,40.464,157.733
C06895=1045.230,303.996,387.773,172.210,40.467,157.734
C06896=1045.238,304.243,387.739,172.214,40.470,157.735
C06897=1045.244,304.491,387.707,172.218,40.473,157.736
C06898=1045.253,304.807,387.664,172.223,40.477,157.737
C06899=1045.262,305.122,387.622,172.227,40.480,157.737
C06900=1045.270,305.438,387.580,172.232,40.484,157.739
C06901=1045.279,305.754,387.538,172.237,40.487,157.740
C06902=1045.286,306.001,387.505,172.240,40.490,157.740
C06903=1045.293,306.249,387.471,172.244,40.493,157.741
C06904=1045.299,306.496,387.438,172.248,40.496,157.742
C06905=1045.307,306.744,387.405,172.252,40.499,157.743
C06906=1045.314,306.991,387.372,172.255,40.501,157.744
C06907=1045.321,307.239,387.339,172.259,40.504,157.744
C06908=1045.327,307.486,387.305,172.263,40.507,157.745
C06909=1045.334,307.735,387.272,172.267,40.510,157.746
C06910=1045.341,307.982,387.239,172.271,40.513,157.747
C06911=1045.348,308.230,387.206,172.275,40.516,157.748
C06912=1045.355,308.478,387.172,172.278,40.519,157.748
C06913=1045.362,308.725,387.140,172.281,40.521,157.749
C06914=1045.369,308.973,387.106,172.285,40.525,157.750
C06915=1045.376,309.220,387.072,172.289,40.527,157.751
C06916=1045.382,309.468,387.039,172.293,40.530,157.752
C06917=1045.390,309.715,387.006,172.297,40.533,157.753
C06918=1045.397,309.963,386.972,172.301,40.536,157.753
C06919=1045.403,310.211,386.939,172.305,40.539,157.754
C06920=1045.410,310.458,386.905,172.309,40.542,157.755
C06921=1045.418,310.706,386.871,172.312,40.544,157.756
C06922=1045.424,310.954,386.839,172.316,40.548,157.757
C06923=1045.432,311.201,386.805,172.320,40.550,157.758
C06924=1045.439,311.449,386.772,172.324,40.553,157.758
C06925=1045.446,311.696,386.738,172.328,40.556,157.759
C06926=1045.452,311.944,386.705,172.332,40.559,157.760
C06927=1045.460,312.192,386.671,172.336,40.562,157.761
C06928=1045.467,312.439,386.637,172.340,40.565,157.762
C06929=1045.474,312.687,386.603,172.344,40.568,157.763
C06930=1045.480,312.934,386.569,172.348,40.571,157.764
C06931=1045.487,313.182,386.536,172.352,40.574,157.764
C06932=1045.494,313.430,386.501,172.356,40.577,157.765
C06933=1045.500,313.677,386.468,172.360,40.580,157.766
C06934=1045.507,313.925,386.433,172.363,40.583,157.767
C06935=1045.514,314.173,386.399,172.367,40.586,157.768
C06936=1045.520,314.420,386.366,172.371,40.589,157.769
C06937=1045.527,314.668,386.332,172.375,40.592,157.770
C06938=1045.534,314.915,386.298,172.379,40.595,157.770
C06939=1045.540,315.163,386.264,172.383,40.598,157.771
C06940=1045.547,315.410,386.229,172.387,40.602,157.772
C06941=1045.554,315.658,386.195,172.391,40.605,157.773
C06942=1045.561,315.905,386.161,172.395,40.608,157.774
C06943=1045.568,316.153,386.127,172.399,40.611,157.775
C06944=1045.574,316.400,386.093,172.403,40.614,157.776
C06945=1045.581,316.648,386.058,172.407,40.617,157.777
C06946=1045.588,316.895,386.024,172.411,40.620,157.778
C06947=1045.595,317.143,385.990,172.415,40.624,157.779
C06948=1045.602,317.391,385.956,172.419,40.626,157.779
C06949=1045.608,317.638,385.921,172.423,40.629,157.780
C06950=1045.615,317.885,385.887,172.427,40.633,157.781
C06951=1045.622,318.133,385.853,172.431,40.636,157.782
C06952=1045.629,318.380,385.818,172.435,40.639,157.783
C06953=1045.636,318.628,385.784,172.439,40.642,157.784
C06954=1045.644,318.948,385.739,172.444,40.646,157.785
C06955=1045.653,319.269,385.695,172.449,40.650,157.786
C06956=1045.662,319.588,385.651,172.454,40.654,157.787
C06957=1045.671,319.909,385.606,172.460,40.658,157.789
C06958=1045.678,320.156,385.572,172.464,40.661,157.789
C06959=1045.685,320.404,385.537,172.468,40.665,157.790
C06960=1045.692,320.651,385.503,172.472,40.668,157.791
C06961=1045.699,320.899,385.468,172.476,40.671,157.792
C06962=1045.706,321.147,385.433,172.481,40.674,157.793
C06963=1045.713,321.394,385.399,172.485,40.677,157.794
C06964=1045.720,321.642,385.364,172.489,40.681,157.795
C06965=1045.727,321.889,385.330,172.493,40.684,157.796
C06966=1045.734,322.137,385.295,172.497,40.687,157.797
C06967=1045.741,322.384,385.261,172.501,40.690,157.798
C06968=1045.748,322.632,385.226,172.505,40.693,157.799
C06969=1045.755,322.879,385.192,172.509,40.696,157.800
C06970=1045.762,323.126,385.157,172.514,40.699,157.800
C06971=1045.768,323.374,385.122,172.518,40.703,157.802
C06972=1045.776,323.621,385.088,172.522,40.706,157.802
C06973=1045.783,323.869,385.053,172.526,40.709,157.803
C06974=1045.790,324.116,385.019,172.530,40.713,157.804
C06975=1045.796,324.364,384.984,172.534,40.716,157.805
C06976=1045.803,324.611,384.949,172.539,40.719,157.806
C06977=1045.811,324.859,384.914,172.543,40.722,157.807
C06978=1045.818,325.106,384.879,172.547,40.725,157.808
C06979=1045.825,325.354,384.845,172.551,40.728,157.809
C06980=1045.832,325.601,384.810,172.555,40.732,157.810
C06981=1045.839,325.849,384.774,172.560,40.735,157.811
C06982=1045.846,326.096,384.740,172.564,40.738,157.812
C06983=1045.854,326.344,384.704,172.568,40.741,157.813
C06984=1045.861,326.591,384.670,172.572,40.745,157.814
C06985=1045.868,326.839,384.635,172.577,40.748,157.815
C06986=1045.874,327.086,384.600,172.581,40.751,157.816
C06987=1045.883,327.334,384.565,172.585,40.754,157.817
C06988=1045.889,327.581,384.530,172.589,40.758,157.817
C06989=1045.897,327.828,384.496,172.594,40.761,157.818
C06990=1045.904,328.076,384.461,172.598,40.764,157.820
C06991=1045.911,328.324,384.425,172.602,40.768,157.820
C06992=1045.919,328.571,384.391,172.606,40.771,157.821
C06993=1045.925,328.818,384.355,172.611,40.774,157.822
C06994=1045.933,329.066,384.320,172.615,40.777,157.823
C06995=1045.940,329.313,384.285,172.620,40.781,157.824
C06996=1045.947,329.560,384.250,172.625,40.784,157.825
C06997=1045.954,329.807,384.214,172.629,40.787,157.826
C06998=1045.961,330.055,384.179,172.633,40.791,157.827
C06999=1045.968,330.303,384.144,172.637,40.794,157.828
C07000=1045.975,330.550,384.108,172.642,40.798,157.829
C07001=1045.982,330.797,384.073,172.646,40.801,157.830
C07002=1045.989,331.045,384.037,172.650,40.805,157.831
C07003=1045.996,331.292,384.002,172.654,40.808,157.832
C07004=1046.003,331.539,383.966,172.659,40.812,157.833
C07005=1046.011,331.787,383.931,172.663,40.815,157.834
C07006=1046.018,332.034,383.895,172.668,40.819,157.835
C07007=1046.024,332.281,383.860,172.673,40.822,157.836
C07008=1046.032,332.529,383.824,172.677,40.825,157.837
C07009=1046.039,332.776,383.788,172.681,40.829,157.838
C07010=1046.047,333.091,383.743,172.687,40.833,157.840
C07011=1046.057,333.407,383.697,172.693,40.837,157.841
C07012=1046.065,333.722,383.652,172.698,40.842,157.842
C07013=1046.075,334.037,383.606,172.704,40.847,157.844
C07014=1046.082,334.285,383.571,172.709,40.850,157.845
C07015=1046.089,334.532,383.535,172.713,40.853,157.846
C07016=1046.096,334.779,383.500,172.717,40.857,157.847
C07017=1046.104,335.027,383.464,172.722,40.860,157.848
C07018=1046.111,335.274,383.428,172.726,40.864,157.849
C07019=1046.118,335.522,383.392,172.731,40.868,157.850
C07020=1046.125,335.768,383.356,172.736,40.871,157.851
C07021=1046.132,336.016,383.320,172.740,40.874,157.852
C07022=1046.139,336.264,383.284,172.745,40.878,157.853
C07023=1046.147,336.511,383.248,172.749,40.882,157.854
C07024=1046.154,336.758,383.212,172.753,40.886,157.855
C07025=1046.161,337.005,383.176,172.759,40.889,157.856
C07026=1046.167,337.253,383.140,172.763,40.892,157.857
C07027=1046.175,337.500,383.104,172.768,40.896,157.858
C07028=1046.181,337.747,383.068,172.772,40.900,157.859
C07029=1046.189,337.995,383.032,172.776,40.904,157.860
C07030=1046.196,338.242,382.996,172.781,40.907,157.862
C07031=1046.203,338.489,382.959,172.786,40.911,157.863
C07032=1046.210,338.736,382.923,172.791,40.915,157.864
C07033=1046.218,338.983,382.887,172.795,40.918,157.865
C07034=1046.225,339.230,382.851,172.800,40.922,157.866
C07035=1046.232,339.478,382.814,172.804,40.926,157.867
C07036=1046.240,339.725,382.778,172.810,40.929,157.868
C07037=1046.247,339.972,382.742,172.814,40.932,157.869
C07038=1046.254,340.220,382.705,172.818,40.936,157.870
C07039=1046.261,340.467,382.669,172.823,40.940,157.871
C07040=1046.268,340.714,382.633,172.827,40.944,157.872
C07041=1046.275,340.962,382.596,172.833,40.948,157.874
C07042=1046.283,341.209,382.560,172.837,40.952,157.875
C07043=1046.290,341.456,382.524,172.842,40.955,157.876
C07044=1046.297,341.704,382.488,172.846,40.959,157.877
C07045=1046.305,341.951,382.451,172.852,40.963,157.878
C07046=1046.311,342.198,382.414,172.856,40.966,157.879
C07047=1046.319,342.445,382.378,172.861,40.970,157.880
C07048=1046.326,342.693,382.341,172.865,40.974,157.881
C07049=1046.333,342.939,382.305,172.870,40.977,157.882
C07050=1046.340,343.187,382.268,172.875,40.982,157.884
C07051=1046.348,343.434,382.232,172.880,40.985,157.885
C07052=1046.355,343.681,382.194,172.885,40.989,157.886
C07053=1046.362,343.928,382.158,172.890,40.992,157.887
C07054=1046.369,344.175,382.121,172.895,40.997,157.888
C07055=1046.376,344.423,382.084,172.899,41.000,157.889
C07056=1046.384,344.670,382.048,172.904,41.004,157.890
C07057=1046.391,344.917,382.010,172.909,41.008,157.892
C07058=1046.398,345.164,381.974,172.914,41.012,157.893
C07059=1046.406,345.411,381.937,172.918,41.016,157.894
C07060=1046.412,345.659,381.900,172.924,41.020,157.895
C07061=1046.420,345.906,381.863,172.929,41.023,157.896
C07062=1046.428,346.153,381.825,172.933,41.028,157.897
C07063=1046.435,346.400,381.790,172.938,41.031,157.899
C07064=1046.442,346.647,381.752,172.943,41.035,157.900
C07065=1046.449,346.894,381.715,172.948,41.039,157.901
C07066=1046.458,347.206,381.669,172.954,41.044,157.902
C07067=1046.468,347.518,381.622,172.960,41.049,157.904
C07068=1046.477,347.829,381.575,172.967,41.054,157.905
C07069=1046.486,348.140,381.528,172.973,41.059,157.907
C07070=1046.493,348.387,381.491,172.978,41.063,157.908
C07071=1046.501,348.634,381.454,172.982,41.067,157.909
C07072=1046.508,348.882,381.417,172.988,41.071,157.910
C07073=1046.515,349.129,381.379,172.993,41.075,157.912
C07074=1046.523,349.376,381.342,172.997,41.079,157.913
C07075=1046.531,349.623,381.305,173.003,41.083,157.914
C07076=1046.538,349.870,381.267,173.008,41.087,157.915
C07077=1046.545,350.117,381.230,173.013,41.091,157.916
C07078=1046.553,350.364,381.193,173.018,41.095,157.918
C07079=1046.560,350.611,381.155,173.023,41.099,157.919
C07080=1046.568,350.858,381.118,173.029,41.103,157.920
C07081=1046.575,351.105,381.080,173.033,41.107,157.921
C07082=1046.582,351.352,381.043,173.038,41.111,157.922
C07083=1046.589,351.599,381.005,173.044,41.115,157.924
C07084=1046.597,351.847,380.968,173.048,41.119,157.925
C07085=1046.604,352.094,380.930,173.054,41.124,157.926
C07086=1046.611,352.341,380.893,173.059,41.128,157.928
C07087=1046.619,352.587,380.854,173.063,41.132,157.929
C07088=1046.626,352.835,380.817,173.069,41.136,157.930
C07089=1046.634,353.082,380.779,173.074,41.140,157.931
C07090=1046.641,353.329,380.741,173.080,41.144,157.933
C07091=1046.649,353.576,380.703,173.084,41.148,157.934
C07092=1046.657,353.823,380.666,173.089,41.152,157.935
C07093=1046.664,354.070,380.629,173.095,41.156,157.936
C07094=1046.671,354.316,380.591,173.100,41.161,157.938
C07095=1046.679,354.564,380.553,173.106,41.165,157.939
C07096=1046.686,354.811,380.515,173.110,41.170,157.940
C07097=1046.694,355.058,380.477,173.116,41.174,157.941
C07098=1046.701,355.305,380.439,173.121,41.178,157.943
C07099=1046.709,355.552,380.401,173.126,41.182,157.944
C07100=1046.716,355.799,380.364,173.132,41.186,157.945
C07101=1046.724,356.046,380.325,173.136,41.190,157.947
C07102=1046.731,356.293,380.287,173.142,41.195,157.948
C07103=1046.739,356.540,380.249,173.147,41.199,157.949
C07104=1046.746,356.787,380.212,173.153,41.203,157.951
C07105=1046.754,357.034,380.173,173.158,41.208,157.952
C07106=1046.762,357.281,380.136,173.164,41.212,157.953
C07107=1046.768,357.528,380.097,173.168,41.216,157.954
C07108=1046.776,357.774,380.058,173.174,41.221,157.956
C07109=1046.784,358.022,380.021,173.179,41.225,157.957
C07110=1046.791,358.269,379.982,173.185,41.229,157.958
C07111=1046.799,358.515,379.944,173.190,41.234,157.960
C07112=1046.807,358.763,379.905,173.196,41.238,157.961
C07113=1046.814,359.010,379.867,173.201,41.242,157.962
C07114=1046.821,359.256,379.829,173.206,41.247,157.964
C07115=1046.829,359.504,379.790,173.211,41.251,157.965
C07116=1046.837,359.750,379.752,173.217,41.256,157.966
C07117=1046.844,359.997,379.714,173.222,41.260,157.968
C07118=1046.852,360.244,379.675,173.228,41.264,157.969
C07119=1046.859,360.491,379.637,173.233,41.268,157.970
C07120=1046.867,360.738,379.598,173.239,41.273,157.972
C07121=1046.875,360.984,379.560,173.244,41.277,157.973
C07122=1046.884,361.302,379.510,173.251,41.283,157.975
C07123=1046.894,361.618,379.461,173.258,41.289,157.977
C07124=1046.904,361.936,379.412,173.265,41.294,157.978
C07125=1046.914,362.253,379.361,173.273,41.301,157.980
C07126=1046.921,362.500,379.323,173.278,41.305,157.982
C07127=1046.930,362.747,379.284,173.284,41.310,157.983
C07128=1046.937,362.993,379.245,173.289,41.314,157.984
C07129=1046.945,363.240,379.206,173.295,41.319,157.986
C07130=1046.952,363.487,379.167,173.300,41.323,157.987
C07131=1046.960,363.734,379.129,173.306,41.328,157.989
C07132=1046.967,363.980,379.089,173.312,41.332,157.990
C07133=1046.975,364.228,379.050,173.317,41.337,157.991
C07134=1046.982,364.474,379.011,173.323,41.342,157.993
C07135=1046.990,364.721,378.972,173.329,41.346,157.994
C07136=1046.997,364.968,378.933,173.334,41.351,157.996
C07137=1047.006,365.215,378.894,173.340,41.356,157.997
C07138=1047.013,365.462,378.855,173.346,41.360,157.999
C07139=1047.021,365.708,378.816,173.351,41.365,158.000
C07140=1047.028,365.955,378.777,173.357,41.370,158.002
C07141=1047.036,366.201,378.738,173.363,41.374,158.003
C07142=1047.044,366.449,378.699,173.368,41.379,158.004
C07143=1047.051,366.696,378.659,173.374,41.384,158.006
C07144=1047.059,366.942,378.620,173.381,41.388,158.007
C07145=1047.067,367.189,378.581,173.386,41.393,158.009
C07146=1047.075,367.436,378.541,173.392,41.398,158.010
C07147=1047.082,367.682,378.502,173.398,41.403,158.012
C07148=1047.090,367.929,378.463,173.403,41.407,158.013
C07149=1047.098,368.176,378.423,173.409,41.412,158.015
C07150=1047.106,368.423,378.384,173.415,41.417,158.016
C07151=1047.114,368.669,378.344,173.420,41.422,158.018
C07152=1047.121,368.916,378.304,173.426,41.427,158.019
C07153=1047.129,369.163,378.266,173.433,41.432,158.021
C07154=1047.137,369.410,378.226,173.439,41.436,158.022
C07155=1047.146,369.657,378.187,173.444,41.441,158.024
C07156=1047.153,369.903,378.147,173.450,41.446,158.025
C07157=1047.161,370.149,378.108,173.456,41.451,158.027
C07158=1047.169,370.396,378.068,173.463,41.455,158.028
C07159=1047.177,370.643,378.028,173.468,41.461,158.030
C07160=1047.185,370.890,377.988,173.474,41.465,158.031
C07161=1047.193,371.137,377.949,173.480,41.470,158.033
C07162=1047.200,371.383,377.909,173.486,41.475,158.034
C07163=1047.208,371.629,377.870,173.492,41.480,158.036
C07164=1047.216,371.876,377.830,173.498,41.485,158.037
C07165=1047.224,372.123,377.789,173.504,41.490,158.039
C07166=1047.232,372.370,377.749,173.510,41.495,158.041
C07167=1047.240,372.616,377.709,173.516,41.500,158.042
C07168=1047.247,372.863,377.669,173.523,41.506,158.044
C07169=1047.255,373.110,377.629,173.528,41.511,158.045
C07170=1047.263,373.357,377.589,173.534,41.515,158.047
C07171=1047.270,373.602,377.549,173.540,41.521,158.048
C07172=1047.278,373.849,377.509,173.547,41.526,158.050
C07173=1047.287,374.096,377.469,173.553,41.531,158.052
C07174=1047.295,374.342,377.429,173.559,41.536,158.053
C07175=1047.302,374.589,377.389,173.565,41.541,158.055
C07176=1047.310,374.835,377.348,173.571,41.546,158.056
C07177=1047.318,375.082,377.308,173.577,41.551,158.058
C07178=1047.329,375.418,377.253,173.586,41.558,158.060
C07179=1047.340,375.754,377.198,173.594,41.565,158.062
C07180=1047.351,376.092,377.143,173.603,41.572,158.065
C07181=1047.363,376.427,377.088,173.611,41.579,158.067
C07182=1047.371,376.674,377.047,173.617,41.585,158.069
C07183=1047.378,376.921,377.007,173.624,41.590,158.070
C07184=1047.386,377.167,376.967,173.630,41.595,158.072
C07185=1047.394,377.413,376.926,173.636,41.600,158.073
C07186=1047.402,377.659,376.885,173.643,41.605,158.075
C07187=1047.411,377.906,376.844,173.649,41.611,158.077
C07188=1047.419,378.153,376.805,173.656,41.616,158.079
C07189=1047.427,378.400,376.764,173.662,41.621,158.080
C07190=1047.435,378.646,376.723,173.668,41.626,158.082
C07191=1047.443,378.892,376.683,173.675,41.632,158.084
C07192=1047.451,379.139,376.642,173.681,41.637,158.085
C07193=1047.459,379.385,376.601,173.688,41.643,158.087
C07194=1047.467,379.632,376.560,173.694,41.648,158.089
C07195=1047.475,379.878,376.520,173.701,41.653,158.090
C07196=1047.483,380.125,376.478,173.707,41.659,158.092
C07197=1047.491,380.372,376.437,173.714,41.664,158.094
C07198=1047.500,380.617,376.396,173.720,41.670,158.096
C07199=1047.508,380.864,376.356,173.727,41.675,158.097
C07200=1047.516,381.111,376.314,173.733,41.681,158.099
C07201=1047.524,381.357,376.273,173.740,41.686,158.101
C07202=1047.532,381.603,376.232,173.746,41.691,158.102
C07203=1047.541,381.850,376.191,173.753,41.697,158.104
C07204=1047.548,382.096,376.150,173.759,41.703,158.106
C07205=1047.556,382.342,376.108,173.766,41.708,158.108
C07206=1047.565,382.589,376.067,173.772,41.714,158.110
C07207=1047.572,382.835,376.025,173.779,41.720,158.111
C07208=1047.581,383.082,375.984,173.786,41.725,158.113
C07209=1047.589,383.328,375.943,173.792,41.730,158.115
C07210=1047.597,383.574,375.902,173.799,41.736,158.117
C07211=1047.606,383.821,375.860,173.806,41.742,158.118
C07212=1047.614,384.067,375.819,173.813,41.747,158.120
C07213=1047.622,384.314,375.777,173.819,41.753,158.122
C07214=1047.630,384.559,375.736,173.826,41.759,158.124
C07215=1047.639,384.806,375.695,173.832,41.765,158.126
C07216=1047.646,385.052,375.653,173.839,41.770,158.127
C07217=1047.655,385.299,375.611,173.847,41.776,158.129
C07218=1047.664,385.546,375.570,173.853,41.781,158.131
C07219=1047.672,385.792,375.528,173.860,41.787,158.133
C07220=1047.681,386.038,375.486,173.867,41.793,158.135
C07221=1047.689,386.284,375.445,173.873,41.799,158.137
C07222=1047.697,386.530,375.403,173.880,41.804,158.138
C07223=1047.706,386.777,375.361,173.888,41.810,158.140
C07224=1047.714,387.023,375.320,173.895,41.816,158.142
C07225=1047.722,387.270,375.278,173.901,41.822,158.144
C07226=1047.731,387.516,375.236,173.908,41.828,158.146
C07227=1047.739,387.762,375.195,173.915,41.833,158.148
C07228=1047.748,388.008,375.153,173.922,41.839,158.150
C07229=1047.757,388.255,375.111,173.929,41.845,158.152
C07230=1047.766,388.500,375.069,173.936,41.851,158.154
C07231=1047.773,388.746,375.027,173.943,41.857,158.155
C07232=1047.782,388.993,374.985,173.951,41.863,158.157
C07233=1047.791,389.239,374.943,173.957,41.869,158.159
C07234=1047.799,389.482,374.901,173.964,41.874,158.161
C07235=1047.807,389.726,374.860,173.972,41.880,158.163
C07236=1047.816,389.969,374.818,173.979,41.887,158.165
C07237=1047.824,390.213,374.776,173.985,41.893,158.167
C07238=1047.833,390.456,374.734,173.992,41.898,158.169
C07239=1047.840,390.700,374.693,174.000,41.904,158.171
C07240=1047.849,390.943,374.650,174.007,41.910,158.173
C07241=1047.858,391.187,374.608,174.014,41.917,158.175
C07242=1047.871,391.561,374.544,174.025,41.926,158.178
C07243=1047.884,391.936,374.479,174.036,41.935,158.181
C07244=1047.896,392.311,374.414,174.047,41.944,158.184
C07245=1047.910,392.686,374.349,174.058,41.954,158.187
C07246=1047.918,392.932,374.307,174.065,41.960,158.189
C07247=1047.927,393.178,374.264,174.073,41.966,158.191
C07248=1047.936,393.424,374.221,174.080,41.972,158.193
C07249=1047.944,393.670,374.178,174.088,41.979,158.195
C07250=1047.953,393.916,374.135,174.095,41.985,158.197
C07251=1047.961,394.163,374.093,174.103,41.991,158.199
C07252=1047.970,394.409,374.050,174.110,41.997,158.201
C07253=1047.979,394.655,374.007,174.118,42.004,158.203
C07254=1047.987,394.901,373.964,174.125,42.010,158.205
C07255=1047.996,395.147,373.921,174.133,42.017,158.207
C07256=1048.004,395.393,373.878,174.140,42.023,158.209
C07257=1048.013,395.639,373.835,174.148,42.029,158.212
C07258=1048.022,395.885,373.793,174.155,42.035,158.214
C07259=1048.031,396.131,373.749,174.163,42.042,158.216
C07260=1048.040,396.377,373.706,174.170,42.048,158.218
C07261=1048.048,396.623,373.663,174.178,42.055,158.220
C07262=1048.057,396.869,373.620,174.185,42.062,158.222
C07263=1048.066,397.114,373.576,174.193,42.068,158.224
C07264=1048.074,397.360,373.533,174.200,42.074,158.226
C07265=1048.083,397.607,373.490,174.209,42.081,158.228
C07266=1048.092,397.853,373.446,174.217,42.087,158.231
C07267=1048.101,398.099,373.403,174.224,42.094,158.233
C07268=1048.109,398.344,373.359,174.232,42.101,158.235
C07269=1048.119,398.591,373.316,174.240,42.107,158.237
C07270=1048.127,398.836,373.272,174.247,42.114,158.239
C07271=1048.136,399.082,373.229,174.255,42.121,158.242
C07272=1048.145,399.328,373.185,174.263,42.127,158.244
C07273=1048.154,399.574,373.142,174.271,42.134,158.246
C07274=1048.162,399.821,373.097,174.279,42.141,158.248
C07275=1048.171,400.066,373.053,174.287,42.147,158.250
C07276=1048.180,400.312,373.010,174.294,42.154,158.253
C07277=1048.189,400.559,372.966,174.303,42.161,158.255
C07278=1048.198,400.804,372.922,174.311,42.167,158.257
C07279=1048.207,401.050,372.878,174.318,42.174,158.259
C07280=1048.216,401.296,372.835,174.326,42.181,158.262
